// TwinCAT 3 PLC project mobject_core
// Title: mobject-core
// Company: mobject.io
// Author: mobject dev team
// ProjectVersion: 0.9.0
// ProgramVersion: 3.1.4023.0
// libraries:
//   Tc2_Standard, * (Beckhoff Automation GmbH)
//   Tc2_System, * (Beckhoff Automation GmbH)
//   Tc2_Utilities, * (Beckhoff Automation GmbH)
//   Tc3_DynamicMemory, * (Beckhoff Automation GmbH)
//   Tc3_Module, * (Beckhoff Automation GmbH)
// project tree:
//   Command/By Inheritance/ Command.TcPOU
//   Command/ I_Command.TcIO
//   / Constants.TcGVL
//   Cyclic Instance/By Composition/ AutomaticCyclicCall.TcPOU, ManualCyclicCall.TcPOU
//   Cyclic Instance/By Inheritance/ CyclicInstance.TcPOU
//   Cyclic Instance/ I_CyclicInstance.TcIO (not stored)
//   Functions/Command Feedback/ F_IsError.TcPOU, F_IsDone.TcPOU, F_IsBusy.TcPOU, F_GetErrorId.TcPOU
//   Functions/Converters/BOOL_TO_/ Convert_BOOL_TO_.TcPOU (not stored), Convert_BOOL_TO_BOOL.TcPOU (not stored), Convert_BOOL_TO_BYTE.TcPOU, Convert_BOOL_TO_DATE.TcPOU, Convert_BOOL_TO_DINT.TcPOU, Convert_BOOL_TO_DT.TcPOU (not stored), Convert_BOOL_TO_DWORD.TcPOU (not stored), Convert_BOOL_TO_INT.TcPOU (not stored), Convert_BOOL_TO_LINT.TcPOU (not stored), Convert_BOOL_TO_LREAL.TcPOU, Convert_BOOL_TO_LWORD.TcPOU, Convert_BOOL_TO_REAL.TcPOU (not stored), Convert_BOOL_TO_SINT.TcPOU, Convert_BOOL_TO_STRING.TcPOU (not stored), Convert_BOOL_TO_TIME.TcPOU, Convert_BOOL_TO_TOD.TcPOU, Convert_BOOL_TO_UDINT.TcPOU (not stored), Convert_BOOL_TO_UINT.TcPOU, Convert_BOOL_TO_ULINT.TcPOU, Convert_BOOL_TO_USINT.TcPOU (not stored), Convert_BOOL_TO_WORD.TcPOU
//   Functions/Converters/BYTE_TO_/ Convert_BYTE_TO_.TcPOU (not stored), Convert_BYTE_TO_BOOL.TcPOU (not stored), Convert_BYTE_TO_BYTE.TcPOU, Convert_BYTE_TO_DATE.TcPOU, Convert_BYTE_TO_DINT.TcPOU (not stored), Convert_BYTE_TO_DT.TcPOU, Convert_BYTE_TO_DWORD.TcPOU (not stored), Convert_BYTE_TO_INT.TcPOU (not stored), Convert_BYTE_TO_LINT.TcPOU (not stored), Convert_BYTE_TO_LREAL.TcPOU, Convert_BYTE_TO_LWORD.TcPOU (not stored), Convert_BYTE_TO_REAL.TcPOU, Convert_BYTE_TO_SINT.TcPOU (not stored), Convert_BYTE_TO_STRING.TcPOU (not stored), Convert_BYTE_TO_TIME.TcPOU, Convert_BYTE_TO_TOD.TcPOU (not stored), Convert_BYTE_TO_UDINT.TcPOU, Convert_BYTE_TO_UINT.TcPOU, Convert_BYTE_TO_ULINT.TcPOU, Convert_BYTE_TO_USINT.TcPOU (not stored), Convert_BYTE_TO_WORD.TcPOU
//   Functions/Converters/DATE_TO_/ Convert_DATE_TO_.TcPOU, Convert_DATE_TO_BOOL.TcPOU, Convert_DATE_TO_BYTE.TcPOU, Convert_DATE_TO_DATE.TcPOU, Convert_DATE_TO_DINT.TcPOU, Convert_DATE_TO_DT.TcPOU (not stored), Convert_DATE_TO_DWORD.TcPOU (not stored), Convert_DATE_TO_INT.TcPOU, Convert_DATE_TO_LINT.TcPOU (not stored), Convert_DATE_TO_LREAL.TcPOU (not stored), Convert_DATE_TO_LWORD.TcPOU (not stored), Convert_DATE_TO_REAL.TcPOU, Convert_DATE_TO_SINT.TcPOU, Convert_DATE_TO_STRING.TcPOU, Convert_DATE_TO_TIME.TcPOU, Convert_DATE_TO_TOD.TcPOU, Convert_DATE_TO_UDINT.TcPOU, Convert_DATE_TO_UINT.TcPOU (not stored), Convert_DATE_TO_ULINT.TcPOU (not stored), Convert_DATE_TO_USINT.TcPOU (not stored), Convert_DATE_TO_WORD.TcPOU
//   Functions/Converters/DINT_TO_/ Convert_DINT_TO_.TcPOU, Convert_DINT_TO_BOOL.TcPOU, Convert_DINT_TO_BYTE.TcPOU, Convert_DINT_TO_DATE.TcPOU (not stored), Convert_DINT_TO_DINT.TcPOU (not stored), Convert_DINT_TO_DT.TcPOU (not stored), Convert_DINT_TO_DWORD.TcPOU, Convert_DINT_TO_INT.TcPOU, Convert_DINT_TO_LINT.TcPOU, Convert_DINT_TO_LREAL.TcPOU (not stored), Convert_DINT_TO_LWORD.TcPOU, Convert_DINT_TO_REAL.TcPOU (not stored), Convert_DINT_TO_SINT.TcPOU, Convert_DINT_TO_STRING.TcPOU, Convert_DINT_TO_TIME.TcPOU (not stored), Convert_DINT_TO_TOD.TcPOU (not stored), Convert_DINT_TO_UDINT.TcPOU, Convert_DINT_TO_UINT.TcPOU (not stored), Convert_DINT_TO_ULINT.TcPOU (not stored), Convert_DINT_TO_USINT.TcPOU, Convert_DINT_TO_WORD.TcPOU
//   Functions/Converters/DT_TO_/ Convert_DT_TO_.TcPOU (not stored), Convert_DT_TO_BOOL.TcPOU, Convert_DT_TO_BYTE.TcPOU, Convert_DT_TO_DATE.TcPOU, Convert_DT_TO_DINT.TcPOU (not stored), Convert_DT_TO_DT.TcPOU (not stored), Convert_DT_TO_DWORD.TcPOU, Convert_DT_TO_INT.TcPOU, Convert_DT_TO_LINT.TcPOU (not stored), Convert_DT_TO_LREAL.TcPOU (not stored), Convert_DT_TO_LWORD.TcPOU, Convert_DT_TO_REAL.TcPOU, Convert_DT_TO_SINT.TcPOU, Convert_DT_TO_STRING.TcPOU, Convert_DT_TO_TIME.TcPOU (not stored), Convert_DT_TO_TOD.TcPOU (not stored), Convert_DT_TO_UDINT.TcPOU, Convert_DT_TO_UINT.TcPOU, Convert_DT_TO_ULINT.TcPOU (not stored), Convert_DT_TO_USINT.TcPOU, Convert_DT_TO_WORD.TcPOU (not stored)
//   Functions/Converters/DWORD_TO_/ Convert_DWORD_TO_.TcPOU, Convert_DWORD_TO_BOOL.TcPOU (not stored), Convert_DWORD_TO_BYTE.TcPOU, Convert_DWORD_TO_DATE.TcPOU, Convert_DWORD_TO_DINT.TcPOU (not stored), Convert_DWORD_TO_DT.TcPOU (not stored), Convert_DWORD_TO_DWORD.TcPOU, Convert_DWORD_TO_INT.TcPOU, Convert_DWORD_TO_LINT.TcPOU, Convert_DWORD_TO_LREAL.TcPOU (not stored), Convert_DWORD_TO_LWORD.TcPOU, Convert_DWORD_TO_REAL.TcPOU, Convert_DWORD_TO_SINT.TcPOU (not stored), Convert_DWORD_TO_STRING.TcPOU (not stored), Convert_DWORD_TO_TIME.TcPOU (not stored), Convert_DWORD_TO_TOD.TcPOU, Convert_DWORD_TO_UDINT.TcPOU, Convert_DWORD_TO_UINT.TcPOU, Convert_DWORD_TO_ULINT.TcPOU, Convert_DWORD_TO_USINT.TcPOU (not stored), Convert_DWORD_TO_WORD.TcPOU
//   Functions/Converters/INT_TO_/ Convert_INT_TO_.TcPOU (not stored), Convert_INT_TO_BOOL.TcPOU (not stored), Convert_INT_TO_BYTE.TcPOU, Convert_INT_TO_DATE.TcPOU (not stored), Convert_INT_TO_DINT.TcPOU (not stored), Convert_INT_TO_DT.TcPOU, Convert_INT_TO_DWORD.TcPOU (not stored), Convert_INT_TO_INT.TcPOU (not stored), Convert_INT_TO_LINT.TcPOU (not stored), Convert_INT_TO_LREAL.TcPOU, Convert_INT_TO_LWORD.TcPOU, Convert_INT_TO_REAL.TcPOU (not stored), Convert_INT_TO_SINT.TcPOU (not stored), Convert_INT_TO_STRING.TcPOU, Convert_INT_TO_TIME.TcPOU (not stored), Convert_INT_TO_TOD.TcPOU, Convert_INT_TO_UDINT.TcPOU (not stored), Convert_INT_TO_UINT.TcPOU (not stored), Convert_INT_TO_ULINT.TcPOU (not stored), Convert_INT_TO_USINT.TcPOU (not stored), Convert_INT_TO_WORD.TcPOU (not stored)
//   Functions/Converters/LINT_TO/ Convert_LINT_TO_.TcPOU (not stored), Convert_LINT_TO_BOOL.TcPOU (not stored), Convert_LINT_TO_BYTE.TcPOU (not stored), Convert_LINT_TO_DATE.TcPOU, Convert_LINT_TO_DINT.TcPOU (not stored), Convert_LINT_TO_DT.TcPOU (not stored), Convert_LINT_TO_DWORD.TcPOU, Convert_LINT_TO_INT.TcPOU (not stored), Convert_LINT_TO_LINT.TcPOU (not stored), Convert_LINT_TO_LREAL.TcPOU (not stored), Convert_LINT_TO_LWORD.TcPOU, Convert_LINT_TO_REAL.TcPOU, Convert_LINT_TO_SINT.TcPOU, Convert_LINT_TO_STRING.TcPOU (not stored), Convert_LINT_TO_TIME.TcPOU, Convert_LINT_TO_TOD.TcPOU (not stored), Convert_LINT_TO_UDINT.TcPOU, Convert_LINT_TO_UINT.TcPOU, Convert_LINT_TO_ULINT.TcPOU, Convert_LINT_TO_USINT.TcPOU (not stored), Convert_LINT_TO_WORD.TcPOU
//   Functions/Converters/LREAL_TO_/ Convert_LREAL_TO_.TcPOU, Convert_LREAL_TO_BOOL.TcPOU, Convert_LREAL_TO_BYTE.TcPOU, Convert_LREAL_TO_DATE.TcPOU, Convert_LREAL_TO_DINT.TcPOU (not stored), Convert_LREAL_TO_DT.TcPOU, Convert_LREAL_TO_DWORD.TcPOU, Convert_LREAL_TO_INT.TcPOU, Convert_LREAL_TO_LINT.TcPOU (not stored), Convert_LREAL_TO_LREAL.TcPOU (not stored), Convert_LREAL_TO_LWORD.TcPOU, Convert_LREAL_TO_REAL.TcPOU (not stored), Convert_LREAL_TO_SINT.TcPOU (not stored), Convert_LREAL_TO_STRING.TcPOU (not stored), Convert_LREAL_TO_TIME.TcPOU, Convert_LREAL_TO_TOD.TcPOU (not stored), Convert_LREAL_TO_UDINT.TcPOU (not stored), Convert_LREAL_TO_UINT.TcPOU, Convert_LREAL_TO_ULINT.TcPOU, Convert_LREAL_TO_USINT.TcPOU, Convert_LREAL_TO_WORD.TcPOU
//   Functions/Converters/LWORD_TO_/ Convert_LWORD_TO_.TcPOU (not stored), Convert_LWORD_TO_BOOL.TcPOU, Convert_LWORD_TO_BYTE.TcPOU (not stored), Convert_LWORD_TO_DATE.TcPOU (not stored), Convert_LWORD_TO_DINT.TcPOU (not stored), Convert_LWORD_TO_DT.TcPOU (not stored), Convert_LWORD_TO_DWORD.TcPOU (not stored), Convert_LWORD_TO_INT.TcPOU (not stored), Convert_LWORD_TO_LINT.TcPOU, Convert_LWORD_TO_LREAL.TcPOU (not stored), Convert_LWORD_TO_LWORD.TcPOU (not stored), Convert_LWORD_TO_REAL.TcPOU (not stored), Convert_LWORD_TO_SINT.TcPOU, Convert_LWORD_TO_STRING.TcPOU, Convert_LWORD_TO_TIME.TcPOU, Convert_LWORD_TO_TOD.TcPOU (not stored), Convert_LWORD_TO_UDINT.TcPOU, Convert_LWORD_TO_UINT.TcPOU, Convert_LWORD_TO_ULINT.TcPOU (not stored), Convert_LWORD_TO_USINT.TcPOU, Convert_LWORD_TO_WORD.TcPOU (not stored)
//   Functions/Converters/REAL_TO_/ Convert_REAL_TO_.TcPOU, Convert_REAL_TO_BOOL.TcPOU (not stored), Convert_REAL_TO_BYTE.TcPOU, Convert_REAL_TO_DATE.TcPOU, Convert_REAL_TO_DINT.TcPOU, Convert_REAL_TO_DT.TcPOU (not stored), Convert_REAL_TO_DWORD.TcPOU, Convert_REAL_TO_INT.TcPOU (not stored), Convert_REAL_TO_LINT.TcPOU, Convert_REAL_TO_LREAL.TcPOU (not stored), Convert_REAL_TO_LWORD.TcPOU, Convert_REAL_TO_REAL.TcPOU (not stored), Convert_REAL_TO_SINT.TcPOU (not stored), Convert_REAL_TO_STRING.TcPOU, Convert_REAL_TO_TIME.TcPOU (not stored), Convert_REAL_TO_TOD.TcPOU (not stored), Convert_REAL_TO_UDINT.TcPOU (not stored), Convert_REAL_TO_UINT.TcPOU (not stored), Convert_REAL_TO_ULINT.TcPOU (not stored), Convert_REAL_TO_USINT.TcPOU (not stored), Convert_REAL_TO_WORD.TcPOU (not stored)
//   Functions/Converters/SINT_TO_/ Convert_SINT_TO_.TcPOU (not stored), Convert_SINT_TO_BOOL.TcPOU (not stored), Convert_SINT_TO_BYTE.TcPOU (not stored), Convert_SINT_TO_DATE.TcPOU (not stored), Convert_SINT_TO_DINT.TcPOU (not stored), Convert_SINT_TO_DT.TcPOU (not stored), Convert_SINT_TO_DWORD.TcPOU (not stored), Convert_SINT_TO_INT.TcPOU (not stored), Convert_SINT_TO_LINT.TcPOU (not stored), Convert_SINT_TO_LREAL.TcPOU (not stored), Convert_SINT_TO_LWORD.TcPOU (not stored), Convert_SINT_TO_REAL.TcPOU (not stored), Convert_SINT_TO_SINT.TcPOU (not stored), Convert_SINT_TO_STRING.TcPOU (not stored), Convert_SINT_TO_TIME.TcPOU (not stored), Convert_SINT_TO_TOD.TcPOU (not stored), Convert_SINT_TO_UDINT.TcPOU (not stored), Convert_SINT_TO_UINT.TcPOU (not stored), Convert_SINT_TO_ULINT.TcPOU (not stored), Convert_SINT_TO_USINT.TcPOU (not stored), Convert_SINT_TO_WORD.TcPOU (not stored)
//   Functions/Converters/STRING_TO_/ Convert_STRING_TO_.TcPOU (not stored), Convert_STRING_TO_BOOL.TcPOU (not stored), Convert_STRING_TO_BYTE.TcPOU (not stored), Convert_STRING_TO_DATE.TcPOU (not stored), Convert_STRING_TO_DINT.TcPOU (not stored), Convert_STRING_TO_DT.TcPOU (not stored), Convert_STRING_TO_DWORD.TcPOU (not stored), Convert_STRING_TO_INT.TcPOU (not stored), Convert_STRING_TO_LINT.TcPOU (not stored), Convert_STRING_TO_LREAL.TcPOU (not stored), Convert_STRING_TO_LWORD.TcPOU (not stored), Convert_STRING_TO_REAL.TcPOU (not stored), Convert_STRING_TO_SINT.TcPOU (not stored), Convert_STRING_TO_STRING.TcPOU (not stored), Convert_STRING_TO_TIME.TcPOU (not stored), Convert_STRING_TO_TOD.TcPOU (not stored), Convert_STRING_TO_UDINT.TcPOU (not stored), Convert_STRING_TO_UINT.TcPOU (not stored), Convert_STRING_TO_ULINT.TcPOU (not stored), Convert_STRING_TO_USINT.TcPOU (not stored), Convert_STRING_TO_WORD.TcPOU (not stored)
//   Functions/Converters/TIME_TO_/ Convert_TIME_TO_.TcPOU (not stored), Convert_TIME_TO_BOOL.TcPOU (not stored), Convert_TIME_TO_BYTE.TcPOU (not stored), Convert_TIME_TO_DATE.TcPOU (not stored), Convert_TIME_TO_DINT.TcPOU (not stored), Convert_TIME_TO_DT.TcPOU (not stored), Convert_TIME_TO_DWORD.TcPOU (not stored), Convert_TIME_TO_INT.TcPOU (not stored), Convert_TIME_TO_LINT.TcPOU (not stored), Convert_TIME_TO_LREAL.TcPOU (not stored), Convert_TIME_TO_LWORD.TcPOU (not stored), Convert_TIME_TO_REAL.TcPOU (not stored), Convert_TIME_TO_SINT.TcPOU (not stored), Convert_TIME_TO_STRING.TcPOU (not stored), Convert_TIME_TO_TIME.TcPOU (not stored), Convert_TIME_TO_TOD.TcPOU (not stored), Convert_TIME_TO_UDINT.TcPOU (not stored), Convert_TIME_TO_UINT.TcPOU (not stored), Convert_TIME_TO_ULINT.TcPOU (not stored), Convert_TIME_TO_USINT.TcPOU (not stored), Convert_TIME_TO_WORD.TcPOU (not stored)
//   Functions/Converters/TOD_TO_/ Convert_TOD_TO_.TcPOU (not stored), Convert_TOD_TO_BOOL.TcPOU (not stored), Convert_TOD_TO_BYTE.TcPOU (not stored), Convert_TOD_TO_DATE.TcPOU (not stored), Convert_TOD_TO_DINT.TcPOU (not stored), Convert_TOD_TO_DT.TcPOU (not stored), Convert_TOD_TO_DWORD.TcPOU (not stored), Convert_TOD_TO_INT.TcPOU (not stored), Convert_TOD_TO_LINT.TcPOU (not stored), Convert_TOD_TO_LREAL.TcPOU (not stored), Convert_TOD_TO_LWORD.TcPOU (not stored), Convert_TOD_TO_REAL.TcPOU (not stored), Convert_TOD_TO_SINT.TcPOU (not stored), Convert_TOD_TO_STRING.TcPOU (not stored), Convert_TOD_TO_TIME.TcPOU (not stored), Convert_TOD_TO_TOD.TcPOU (not stored), Convert_TOD_TO_UDINT.TcPOU (not stored), Convert_TOD_TO_UINT.TcPOU (not stored), Convert_TOD_TO_ULINT.TcPOU (not stored), Convert_TOD_TO_USINT.TcPOU (not stored), Convert_TOD_TO_WORD.TcPOU (not stored)
//   Functions/Converters/UDINT_TO_/ Convert_UDINT_TO_.TcPOU (not stored), Convert_UDINT_TO_BOOL.TcPOU (not stored), Convert_UDINT_TO_BYTE.TcPOU (not stored), Convert_UDINT_TO_DATE.TcPOU (not stored), Convert_UDINT_TO_DINT.TcPOU (not stored), Convert_UDINT_TO_DT.TcPOU (not stored), Convert_UDINT_TO_DWORD.TcPOU (not stored), Convert_UDINT_TO_INT.TcPOU (not stored), Convert_UDINT_TO_LINT.TcPOU (not stored), Convert_UDINT_TO_LREAL.TcPOU (not stored), Convert_UDINT_TO_LWORD.TcPOU (not stored), Convert_UDINT_TO_REAL.TcPOU (not stored), Convert_UDINT_TO_SINT.TcPOU (not stored), Convert_UDINT_TO_STRING.TcPOU (not stored), Convert_UDINT_TO_TIME.TcPOU (not stored), Convert_UDINT_TO_TOD.TcPOU (not stored), Convert_UDINT_TO_UDINT.TcPOU (not stored), Convert_UDINT_TO_UINT.TcPOU (not stored), Convert_UDINT_TO_ULINT.TcPOU (not stored), Convert_UDINT_TO_USINT.TcPOU (not stored), Convert_UDINT_TO_WORD.TcPOU (not stored)
//   Functions/Converters/UINT_TO_/ Convert_UINT_TO_.TcPOU (not stored), Convert_UINT_TO_BOOL.TcPOU (not stored), Convert_UINT_TO_BYTE.TcPOU (not stored), Convert_UINT_TO_DATE.TcPOU (not stored), Convert_UINT_TO_DINT.TcPOU (not stored), Convert_UINT_TO_DT.TcPOU (not stored), Convert_UINT_TO_DWORD.TcPOU (not stored), Convert_UINT_TO_INT.TcPOU (not stored), Convert_UINT_TO_LINT.TcPOU (not stored), Convert_UINT_TO_LREAL.TcPOU (not stored), Convert_UINT_TO_LWORD.TcPOU (not stored), Convert_UINT_TO_REAL.TcPOU (not stored), Convert_UINT_TO_SINT.TcPOU (not stored), Convert_UINT_TO_STRING.TcPOU (not stored), Convert_UINT_TO_TIME.TcPOU (not stored), Convert_UINT_TO_TOD.TcPOU (not stored), Convert_UINT_TO_UDINT.TcPOU (not stored), Convert_UINT_TO_UINT.TcPOU (not stored), Convert_UINT_TO_ULINT.TcPOU (not stored), Convert_UINT_TO_USINT.TcPOU (not stored), Convert_UINT_TO_WORD.TcPOU (not stored)
//   Functions/Converters/ULINT_TO_/ Convert_ULINT_TO_.TcPOU (not stored), Convert_ULINT_TO_BOOL.TcPOU (not stored), Convert_ULINT_TO_BYTE.TcPOU (not stored), Convert_ULINT_TO_DATE.TcPOU (not stored), Convert_ULINT_TO_DINT.TcPOU (not stored), Convert_ULINT_TO_DT.TcPOU (not stored), Convert_ULINT_TO_DWORD.TcPOU (not stored), Convert_ULINT_TO_INT.TcPOU (not stored), Convert_ULINT_TO_LINT.TcPOU (not stored), Convert_ULINT_TO_LREAL.TcPOU (not stored), Convert_ULINT_TO_LWORD.TcPOU (not stored), Convert_ULINT_TO_REAL.TcPOU (not stored), Convert_ULINT_TO_SINT.TcPOU (not stored), Convert_ULINT_TO_STRING.TcPOU (not stored), Convert_ULINT_TO_TIME.TcPOU (not stored), Convert_ULINT_TO_TOD.TcPOU (not stored), Convert_ULINT_TO_UDINT.TcPOU (not stored), Convert_ULINT_TO_UINT.TcPOU (not stored), Convert_ULINT_TO_ULINT.TcPOU (not stored), Convert_ULINT_TO_USINT.TcPOU (not stored), Convert_ULINT_TO_WORD.TcPOU (not stored)
//   Functions/Converters/USINT_TO_/ Convert_USINT_TO_.TcPOU (not stored), Convert_USINT_TO_BOOL.TcPOU (not stored), Convert_USINT_TO_BYTE.TcPOU (not stored), Convert_USINT_TO_DATE.TcPOU (not stored), Convert_USINT_TO_DINT.TcPOU (not stored), Convert_USINT_TO_DT.TcPOU (not stored), Convert_USINT_TO_DWORD.TcPOU (not stored), Convert_USINT_TO_INT.TcPOU (not stored), Convert_USINT_TO_LINT.TcPOU (not stored), Convert_USINT_TO_LREAL.TcPOU (not stored), Convert_USINT_TO_LWORD.TcPOU (not stored), Convert_USINT_TO_REAL.TcPOU (not stored), Convert_USINT_TO_SINT.TcPOU (not stored), Convert_USINT_TO_STRING.TcPOU (not stored), Convert_USINT_TO_TIME.TcPOU (not stored), Convert_USINT_TO_TOD.TcPOU (not stored), Convert_USINT_TO_UDINT.TcPOU (not stored), Convert_USINT_TO_UINT.TcPOU (not stored), Convert_USINT_TO_ULINT.TcPOU (not stored), Convert_USINT_TO_USINT.TcPOU (not stored), Convert_USINT_TO_WORD.TcPOU (not stored)
//   Functions/Converters/WORD_TO_/ Convert_WORD_TO_.TcPOU (not stored), Convert_WORD_TO_BOOL.TcPOU (not stored), Convert_WORD_TO_BYTE.TcPOU (not stored), Convert_WORD_TO_DATE.TcPOU (not stored), Convert_WORD_TO_DINT.TcPOU (not stored), Convert_WORD_TO_DT.TcPOU (not stored), Convert_WORD_TO_DWORD.TcPOU (not stored), Convert_WORD_TO_INT.TcPOU (not stored), Convert_WORD_TO_LINT.TcPOU (not stored), Convert_WORD_TO_LREAL.TcPOU (not stored), Convert_WORD_TO_LWORD.TcPOU (not stored), Convert_WORD_TO_REAL.TcPOU (not stored), Convert_WORD_TO_SINT.TcPOU (not stored), Convert_WORD_TO_STRING.TcPOU (not stored), Convert_WORD_TO_TIME.TcPOU (not stored), Convert_WORD_TO_TOD.TcPOU (not stored), Convert_WORD_TO_UDINT.TcPOU (not stored), Convert_WORD_TO_UINT.TcPOU (not stored), Convert_WORD_TO_ULINT.TcPOU (not stored), Convert_WORD_TO_USINT.TcPOU (not stored), Convert_WORD_TO_WORD.TcPOU (not stored)
//   Functions/Disposable/ F_SafeRelease.TcPOU
//   _Internal/Collections/ Collection.TcPOU, CollectionNode.TcPOU, I_Collectable.TcIO, I_CollectionNode.TcIO
//   _Internal/CommandFeedback/ CommandFeedback.TcPOU, I_CommandAbortingState.TcIO, I_CommandBusyState.TcIO, I_CommandFeedback.TcIO, I_CommandFeedbackReadWrite.TcIO
//   _Internal/Command/ I_CanReleaseWhenDone.TcIO
//   _Internal/CyclicCallback/Base/ CyclicCallback.TcPOU (not stored)
//   _Internal/CyclicCallback/Interface/ I_CyclicCalled.TcIO (not stored)
//   _Internal/Disposable/ Disposable.TcPOU, I_Disposable.TcIO
//   _Internal/Events/Base/ Event.TcPOU (not stored), I_Event.TcIO (not stored)
//   _Internal/Events/Collections/ SubscriberCollection.TcPOU (not stored)
//   _Internal/Events/Interfaces/ I_Callback.TcIO (not stored), I_Subscriber.TcIO (not stored)
//   _Internal/Functions/Namespace/ ReturnNamespaceFromInstancePath.TcPOU (not stored), ReturnSubSectionFromInstancePath.TcPOU (not stored)
//   _Internal/GlobalInstanceMembership/ GlobalInstanceMembership.TcPOU
//   _Internal/GlobalInstancesMembers/ GlobalInstanceMembers.TcPOU
//   _Internal/GlobalNamespace/ GlobalNamespace.TcPOU
//   _Internal/Instance/Collection/ InstanceCollection.TcPOU (not stored)
//   _Internal/Instance/Events/InstanceAdded/ InstanceAddedEvent.TcPOU (not stored), I_InstanceAddedEvent.TcIO (not stored)
//   _Internal/Instance/Events/InstanceRemoved/ InstanceRemovedEvent.TcPOU (not stored), I_InstanceRemovedEvent.TcIO (not stored)
//   _Internal/Instance/ Instance.TcPOU, I_Instance.TcIO
//   _Internal/Task/Callbacks/ DeregisterInstanceFromTaskCallback.TcPOU (not stored), RegisterInstanceToTaskCallback.TcPOU (not stored)
//   _Internal/Task/Events/TaskCyclicEvent/ I_TaskCyclicEvent.TcIO (not stored), TaskCyclicEvent.TcPOU (not stored)
//   _Internal/Task/Visitors/ I_VisitIntances.TcIO (not stored), RegisterInstancesToTaskVisitor.TcPOU (not stored)
//   Task/ I_Task.TcIO, Task.TcPOU

// ---- Constants.TcGVL
VAR_GLOBAL CONSTANT
	INVALIDPARM : HRESULT := UDINT_TO_DINT(16#9811070B);
	NOT_FOUND : HRESULT := UDINT_TO_DINT(16#9811070C);
	INCOMPATIBLE : HRESULT := UDINT_TO_DINT(16#9811070E);
END_VAR

// ---- Command/I_Command.TcIO
INTERFACE I_Command EXTENDS I_Disposable

METHOD PUBLIC Abort : I_CanReleaseWhenDone
VAR_INPUT
END_VAR
END_METHOD

METHOD PUBLIC Execute : I_CanReleaseWhenDone
VAR_INPUT
	Feedback : REFERENCE TO I_CommandFeedback;
END_VAR
END_METHOD

END_INTERFACE

// ---- _Internal/Collections/I_Collectable.TcIO
INTERFACE I_Collectable EXTENDS __SYSTEM.IQueryInterface

END_INTERFACE

// ---- _Internal/Collections/I_CollectionNode.TcIO
INTERFACE I_CollectionNode

PROPERTY PUBLIC Collectable : I_Collectable
GET
END_GET
END_PROPERTY

METHOD PUBLIC Destroy
VAR_INPUT
END_VAR
END_METHOD

PROPERTY PUBLIC Next : I_CollectionNode
GET
END_GET
SET
END_SET
END_PROPERTY

END_INTERFACE

// ---- _Internal/CommandFeedback/I_CommandAbortingState.TcIO
INTERFACE I_CommandAbortingState

METHOD PUBLIC SetAborted
VAR_INPUT
END_VAR
END_METHOD

METHOD PUBLIC SetError
VAR_INPUT
	ErrorId : UDINT;
END_VAR
END_METHOD

END_INTERFACE

// ---- _Internal/CommandFeedback/I_CommandBusyState.TcIO
INTERFACE I_CommandBusyState

METHOD PUBLIC SetAborting
VAR_INPUT
END_VAR
END_METHOD

METHOD PUBLIC SetDone
VAR_INPUT
END_VAR
END_METHOD

METHOD PUBLIC SetError
VAR_INPUT
	ErrorId : UDINT;
END_VAR
END_METHOD

END_INTERFACE

// ---- _Internal/CommandFeedback/I_CommandFeedback.TcIO
INTERFACE I_CommandFeedback EXTENDS I_Disposable

PROPERTY Aborted : BOOL
GET
END_GET
END_PROPERTY

PROPERTY Aborting : BOOL
GET
END_GET
END_PROPERTY

PROPERTY Busy : BOOL
GET
END_GET
END_PROPERTY

PROPERTY Done : BOOL
GET
END_GET
END_PROPERTY

PROPERTY Error : BOOL
GET
END_GET
END_PROPERTY

PROPERTY PUBLIC ErrorId : UDINT
GET
END_GET
END_PROPERTY

END_INTERFACE

// ---- _Internal/CommandFeedback/I_CommandFeedbackReadWrite.TcIO
INTERFACE I_CommandFeedbackReadWrite EXTENDS I_CommandFeedback, I_CommandBusyState, I_CommandAbortingState

METHOD PUBLIC SetBusy
VAR_INPUT
END_VAR
END_METHOD

END_INTERFACE

// ---- _Internal/Command/I_CanReleaseWhenDone.TcIO
INTERFACE I_CanReleaseWhenDone

METHOD PUBLIC ThenRelease
VAR_INPUT
END_VAR
END_METHOD

END_INTERFACE

// ---- _Internal/Disposable/I_Disposable.TcIO
INTERFACE I_Disposable EXTENDS __SYSTEM.IQueryInterface

METHOD AddReference
VAR_INPUT
END_VAR
END_METHOD

METHOD Release
VAR_INPUT
END_VAR
END_METHOD

END_INTERFACE

// ---- _Internal/Instance/I_Instance.TcIO
INTERFACE I_Instance EXTENDS I_Collectable

PROPERTY PUBLIC NameSpace : STRING
GET
END_GET
END_PROPERTY

METHOD PUBLIC SharesNamespaceWith : BOOL
VAR_INPUT
	OtherInstance : I_Instance;
END_VAR
END_METHOD

END_INTERFACE

// ---- Task/I_Task.TcIO
INTERFACE I_Task EXTENDS I_Instance

METHOD PUBLIC CyclicCall
END_METHOD

METHOD PUBLIC DeregisterInstance
VAR_INPUT
	Instance : I_Instance;
END_VAR
END_METHOD

PROPERTY PUBLIC Index : DINT
GET
END_GET
END_PROPERTY

PROPERTY Info : reference to PlcTaskSystemInfo
GET
END_GET
END_PROPERTY

METHOD PUBLIC IsExecutingThis : BOOL
VAR_INPUT
END_VAR
END_METHOD

PROPERTY PUBLIC OnCyclicCall : I_Event
GET
END_GET
END_PROPERTY

METHOD PUBLIC RegisterInstance
VAR_INPUT
	Instance : I_Instance;
END_VAR
END_METHOD

END_INTERFACE

// ---- Command/By Inheritance/Command.TcPOU
{attribute 'linkalways'} 
{attribute 'no_explicit_call' := 'This FB is a CLASS and must be accessed using methods or properties'}
{attribute 'enable_dynamic_creation'}
FUNCTION_BLOCK ABSTRACT Command EXTENDS Disposable IMPLEMENTS I_CyclicCalled, I_Command, I_CanReleaseWhenDone
VAR
	cyclicCall : ManualCyclicCall(THIS^);
	commandFeedback : I_CommandFeedbackReadWrite;
	commandHasCompleted : BOOL;
	disposeOnceComplete : BOOL;
END_VAR

METHOD PUBLIC Abort : I_CanReleaseWhenDone
VAR_INPUT
END_VAR
Abort := THIS^;

IF IsAborting() THEN
	RETURN;
END_IF

IF HasCompleted() THEN
	RETURN;
END_IF

commandFeedback.SetAborting();

OnAbort(commandFeedback);

IF HasCompleted() THEN
	DisableCyclicCalling();
	CompleteTheCommand();
	RETURN;
END_IF
END_METHOD

METHOD PRIVATE ClearFeedback
VAR_INPUT
END_VAR
commandFeedback.Release();
commandFeedback := 0;
END_METHOD

METHOD PRIVATE CompleteTheCommand
VAR_INPUT
END_VAR
ClearFeedback();

IF disposeOnceComplete THEN
	DisposeCommand();	
END_IF

OnExecuteComplete();

commandHasCompleted := TRUE;
END_METHOD

METHOD PUBLIC CyclicCall
VAR_INPUT
END_VAR
IF IsStillBusyExecuting() THEN
	WhileBusy(commandFeedback);
END_IF

IF IsAborting() THEN
	WhileAborting(commandFeedback);
END_IF

IF NOT HasCompleted() THEN 
	RETURN;
END_IF

DisableCyclicCalling();
CompleteTheCommand();
END_METHOD

METHOD PRIVATE DisableCyclicCalling
cyclicCall.Disable();
END_METHOD

METHOD PRIVATE DisposeCommand
VAR_INPUT
END_VAR
disposeOnceComplete := FALSE;

SUPER^.OnDispose();
END_METHOD

METHOD PRIVATE EnableCyclicCalling
cyclicCall.Enable();
END_METHOD

METHOD PUBLIC Execute : I_CanReleaseWhenDone
VAR_INPUT
	Feedback : REFERENCE TO I_CommandFeedback;
END_VAR
Execute := THIS^;

IF feedback <> 0 THEN 
	feedback.Release();
END_IF

IF IsAlreadyExecuting() THEN

	IF __ISVALIDREF(feedback) THEN
		feedback := commandFeedback;
		feedback.AddReference();
	END_IF
	
	RETURN;
	
END_IF

IF commandFeedback <> 0 THEN 
	commandFeedback.Release();
END_IF

commandFeedback := GetCustomFeedback();

IF commandFeedback = 0 THEN
	commandFeedback := GetStandardFeedback();
END_IF

IF __ISVALIDREF(feedback) THEN
	feedback := commandFeedback;
	feedback.AddReference();
END_IF

commandFeedback.SetBusy();

OnExecute(commandFeedback);

IF HasCompleted() THEN
	CompleteTheCommand();
	RETURN;
END_IF

EnableCyclicCalling();
END_METHOD

METHOD PROTECTED GetCustomFeedback : I_CommandFeedbackReadWrite
VAR
END_VAR
END_METHOD

METHOD PROTECTED GetStandardFeedback : I_CommandFeedbackReadWrite
VAR
	feedback : POINTER TO CommandFeedback;
END_VAR
feedback := __NEW(CommandFeedback);
GetStandardFeedback := feedback^;
END_METHOD

METHOD PRIVATE HasCompleted : BOOL
IF commandFeedback = 0 THEN
	HasCompleted := commandHasCompleted;
	RETURN;
END_IF

HasCompleted := not commandFeedback.Busy;
END_METHOD

METHOD PRIVATE IsAborting : BOOL
IF commandFeedback = 0 THEN
	RETURN;
END_IF

IsAborting := commandFeedback.Aborting;
END_METHOD

METHOD PRIVATE IsAlreadyExecuting : BOOL
IF commandFeedback = 0 THEN
	RETURN;
END_IF

IsAlreadyExecuting := commandFeedback.Busy;
END_METHOD

METHOD PRIVATE IsStillBusyExecuting : BOOL
IF commandFeedback = 0 THEN
	RETURN;
END_IF

IsStillBusyExecuting := commandFeedback.Busy and not commandFeedback.Aborting;
END_METHOD

METHOD PROTECTED OnAbort
VAR_INPUT
	CommandState : I_CommandAbortingState;
END_VAR
// override this method when a command needs time to "abort".
// if your aborting code take more than one cycle to completed then do not SetAborted() here, rather use SetAborted inside WhileAborting.
CommandState.SetAborted();
END_METHOD

METHOD PROTECTED OnDispose
VAR_INPUT
END_VAR
IF IsAlreadyExecuting() THEN 
	disposeOnceComplete := TRUE;
	Abort();
	RETURN;	
END_IF

DisposeCommand();
END_METHOD

METHOD PROTECTED OnExecute
VAR_INPUT
	CommandState : I_CommandBusyState;
END_VAR
END_METHOD

METHOD PROTECTED OnExecuteComplete
VAR_INPUT
END_VAR
END_METHOD

METHOD PUBLIC ThenRelease
VAR_INPUT
END_VAR
IF HasCompleted() THEN
	DisposeCommand();
	RETURN;
END_IF

disposeOnceComplete := true;
END_METHOD

METHOD PROTECTED WhileAborting
VAR_INPUT
	CommandState : I_CommandAbortingState;
END_VAR
// you must override both OnAbort and WhileAborting to use this method.
// if SetAborted has not been called during OnAbort then this method will be cyclically called until you do;
CommandState.SetAborted();
END_METHOD

METHOD PROTECTED ABSTRACT WhileBusy
VAR_INPUT
	CommandState : I_CommandBusyState;
END_VAR
// This will be called cyclically until the command has finished executing.  
// once done use the command below to complete the execute state.
//commandState.SetDone();

// use SetError to cancel the command.
//CommandState.SetError(ErrorID:=0);
END_METHOD

END_FUNCTION_BLOCK

// ---- _Internal/Disposable/Disposable.TcPOU
{attribute 'linkalways'} 
{attribute 'no_explicit_call' := 'This FB is a CLASS and must be accessed using methods or properties'}
{attribute 'enable_dynamic_creation'}
{attribute 'reflection'}
FUNCTION_BLOCK Disposable IMPLEMENTS I_Disposable
VAR
	{attribute 'instance-path'} 
    {attribute 'noinit'} 
	instancePathUsedToCheckIfDynamic : T_MAXSTRING;
	referenceCount : UDINT := 1;
END_VAR

METHOD AddReference
VAR_INPUT
END_VAR
VAR
	debug : UDINT;
END_VAR
referenceCount := referenceCount + 1;

debug := referenceCount;
END_METHOD

METHOD PROTECTED OnDispose
VAR_INPUT
END_VAR
__DELETE(THIS);
END_METHOD

METHOD Release
VAR_INPUT
END_VAR
VAR
	debug : UDINT;
END_VAR
referenceCount := referenceCount - 1;

debug := referenceCount;

IF referenceCount > 0 THEN
	RETURN;
END_IF

OnDispose();
END_METHOD

END_FUNCTION_BLOCK

// ---- _Internal/Instance/Instance.TcPOU
{attribute 'linkalways'} 
{attribute 'no_explicit_call' := 'This FB is a CLASS and must be accessed using methods or properties'}
{attribute 'enable_dynamic_creation'}
{attribute 'reflection'}
FUNCTION_BLOCK Instance IMPLEMENTS I_Instance, I_Collectable
{attribute 'hide_all_locals'}
VAR
	{attribute 'instance-path'} 
    {attribute 'noinit'} 
	instancePath : T_MAXSTRING;
	instanceNamespace : STRING := GetNamespace();
	globalNamespace : GlobalNamespace(THIS^);
END_VAR

METHOD PRIVATE GetNamespace : STRING
IF InstancePathIsFilled() THEN
	GetNamespace := ReturnNamespaceFromInstancePath(instancePath);
	RETURN;
END_IF

IF IsNewObjectDuringInitialization() THEN
	GetNamespace := globalNamespace.GetLastInstanceNamespace();
END_IF
END_METHOD

METHOD PRIVATE InstancePathIsFilled : BOOL
InstancePathIsFilled := instancePath <> '';
END_METHOD

METHOD PRIVATE IsNewObjectDuringInitialization : BOOL
VAR CONSTANT 
	PLC_INIT_PHASE : INT := 0;
END_VAR
IsNewObjectDuringInitialization := GETCURTASKINDEXEX() = PLC_INIT_PHASE;
END_METHOD

PROPERTY PUBLIC NameSpace : STRING
GET
Namespace := instanceNamespace;
END_GET
END_PROPERTY

METHOD PUBLIC SharesNamespaceWith : BOOL
VAR_INPUT
	OtherInstance : I_Instance;
END_VAR
SharesNamespaceWith := (Namespace = OtherInstance.NameSpace);
END_METHOD

END_FUNCTION_BLOCK

// ---- _Internal/GlobalNamespace/GlobalNamespace.TcPOU
{attribute 'linkalways'} 
{attribute 'no_explicit_call' := 'This FB is a CLASS and must be accessed using methods or properties'}
{attribute 'enable_dynamic_creation'}
FUNCTION_BLOCK GlobalNamespace
VAR_STAT // singleton
	lastInstanceNamespace : STRING;
END_VAR

METHOD FB_init : BOOL
VAR_INPUT
	bInitRetains : BOOL; // if TRUE, the retain variables are initialized (warm start / cold start)
	bInCopyCode : BOOL;  // if TRUE, the instance afterwards gets moved into the copy code (online change)
	Instance : I_Instance;
END_VAR
IF Instance.NameSpace = '' THEN
	RETURN;
END_IF

lastInstanceNamespace := Instance.NameSpace;
END_METHOD

METHOD PUBLIC GetLastInstanceNamespace : String
VAR_INPUT
END_VAR
GetLastInstanceNamespace := lastInstanceNamespace;
END_METHOD

END_FUNCTION_BLOCK

// ---- Cyclic Instance/By Composition/ManualCyclicCall.TcPOU
{attribute 'linkalways'} 
{attribute 'no_explicit_call' := 'This FB is a CLASS and must be accessed using methods or properties'}
{attribute 'enable_dynamic_creation'}
FUNCTION_BLOCK ManualCyclicCall EXTENDS Instance IMPLEMENTS I_CyclicInstance
VAR
	membership : GlobalInstanceMembership(THIS^);
	_cyclicInstanceCallback : CyclicCallback(0);
END_VAR

PROPERTY PUBLIC CyclicInstanceCallback : I_Callback
GET
CyclicInstanceCallback := _cyclicInstanceCallback;
END_GET
END_PROPERTY

METHOD PUBLIC Disable
VAR_INPUT
END_VAR
membership.Leave();
END_METHOD

METHOD PUBLIC Enable
VAR_INPUT
END_VAR
membership.Join();
END_METHOD

METHOD FB_init : BOOL
VAR_INPUT
	bInitRetains : BOOL; // if TRUE, the retain variables are initialized (warm start / cold start)
	bInCopyCode : BOOL;  // if TRUE, the instance afterwards gets moved into the copy code (online change)
	Target : I_CyclicCalled;
END_VAR
_cyclicInstanceCallback.Target := Target;
END_METHOD

END_FUNCTION_BLOCK

// ---- _Internal/GlobalInstanceMembership/GlobalInstanceMembership.TcPOU
{attribute 'linkalways'} 
{attribute 'no_explicit_call' := 'This FB is a CLASS and must be accessed using methods or properties'}
{attribute 'enable_dynamic_creation'}
FUNCTION_BLOCK GlobalInstanceMembership
VAR
	self : I_Instance;
	globalInstanceMembers : GlobalInstanceMembers;
END_VAR

METHOD FB_exit : BOOL
VAR_INPUT
	bInCopyCode : BOOL; // if TRUE, the exit method is called for exiting an instance that is copied afterwards (online change).
END_VAR
Leave();
END_METHOD

METHOD FB_init : BOOL
VAR_INPUT
	bInitRetains : BOOL; // if TRUE, the retain variables are initialized (warm start / cold start)
	bInCopyCode : BOOL;  // if TRUE, the instance afterwards gets moved into the copy code (online change)
	Self : I_Instance;
END_VAR
THIS^.self := Self;
END_METHOD

METHOD PUBLIC Join
VAR_INPUT
END_VAR
globalInstanceMembers.AddInstance(Self);
END_METHOD

METHOD PUBLIC Leave
VAR_INPUT
END_VAR
globalInstanceMembers.RemoveInstance(THIS^.self);
END_METHOD

END_FUNCTION_BLOCK

// ---- _Internal/GlobalInstancesMembers/GlobalInstanceMembers.TcPOU
{attribute 'linkalways'} 
{attribute 'no_explicit_call' := 'This FB is a CLASS and must be accessed using methods or properties'}
{attribute 'enable_dynamic_creation'}
FUNCTION_BLOCK GlobalInstanceMembers
VAR_STAT // singleton
	instances : InstanceCollection;
	instanceAddedEvent : InstanceAddedEvent;
	instanceRemovedEvent : InstanceRemovedEvent;
END_VAR

METHOD PUBLIC AddInstance
VAR_INPUT
	Instance : I_Instance;
END_VAR
IF Instance = 0 THEN
	RETURN;
END_IF

instances.Insert(Instance);
instanceAddedEvent.Notify(Instance);
END_METHOD

METHOD PUBLIC ForEachInstance
VAR_INPUT
	Visitor : I_VisitIntances;
END_VAR
VAR
	last : DINT;
	i : DINT;
END_VAR
last := instances.Count - 1;

FOR i := 0 TO last DO
	Visitor.Visit(instances.GetByIndex(i));
END_FOR
END_METHOD

PROPERTY PUBLIC OnInstanceAdded : I_Event
GET
OnInstanceAdded := instanceAddedEvent;
END_GET
END_PROPERTY

PROPERTY PUBLIC OnInstanceRemoved : I_Event
GET
OnInstanceRemoved := InstanceRemovedEvent;
END_GET
END_PROPERTY

METHOD PUBLIC RemoveInstance
VAR_INPUT
	Instance : I_Instance;
END_VAR
IF Instance = 0 THEN
	RETURN;
END_IF

instances.Remove(Instance);
InstanceRemovedEvent.Notify(Instance);
END_METHOD

END_FUNCTION_BLOCK

// ---- _Internal/CommandFeedback/CommandFeedback.TcPOU
{attribute 'linkalways'} 
{attribute 'no_explicit_call' := 'This FB is a CLASS and must be accessed using methods or properties'}
{attribute 'enable_dynamic_creation'}
FUNCTION_BLOCK CommandFeedback EXTENDS Disposable IMPLEMENTS I_CommandFeedbackReadWrite, I_CommandFeedback, I_CommandBusyState, I_CommandAbortingState
VAR
	_busy : BOOL;
	_done : BOOL;
	_aborted : BOOL;
	_aborting : BOOL;
	_error : BOOL;
	_errorId : UDINT;
END_VAR

PROPERTY Aborted : BOOL
GET
Aborted := _aborted;
END_GET
END_PROPERTY

PROPERTY Aborting : BOOL
GET
Aborting := _aborting;
END_GET
END_PROPERTY

PROPERTY Busy : BOOL
GET
Busy := _busy;
END_GET
END_PROPERTY

PROPERTY Done : BOOL
GET
Done := _done;
END_GET
END_PROPERTY

PROPERTY Error : BOOL
GET
Error := _error;
END_GET
END_PROPERTY

PROPERTY PUBLIC ErrorId : UDINT
GET
END_GET
END_PROPERTY

METHOD PUBLIC SetAborted
VAR_INPUT
END_VAR
_busy := FALSE;
_done := FALSE;
_aborted := TRUE;
_aborting := FALSE;
_error := FALSE;
_errorId := 0;
END_METHOD

METHOD PUBLIC SetAborting
VAR_INPUT
END_VAR
IF NOT Busy THEN
	SetAborted();
	RETURN;
END_IF

_busy := TRUE;
_done := FALSE;
_aborted := FALSE;
_aborting := TRUE;
_error := FALSE;
_errorId := 0;
END_METHOD

METHOD PUBLIC SetBusy
VAR_INPUT
END_VAR
_busy := TRUE;
_done := FALSE;
_aborted := FALSE;
_aborting := FALSE;
_error := FALSE;
_errorId := 0;
END_METHOD

METHOD PUBLIC SetDone
VAR_INPUT
END_VAR
_busy := FALSE;
_done := TRUE;
_aborted := FALSE;
_aborting := FALSE;
_error := FALSE;
_errorId := 0;
END_METHOD

METHOD PUBLIC SetError
VAR_INPUT
	ErrorId : UDINT;
END_VAR
_busy := FALSE;
_done := FALSE;
_aborted := FALSE;
_aborting := FALSE;
_error := TRUE;
_errorId := ErrorId;
END_METHOD

END_FUNCTION_BLOCK

// ---- Cyclic Instance/By Composition/AutomaticCyclicCall.TcPOU
{attribute 'linkalways'} 
{attribute 'no_explicit_call' := 'This FB is a CLASS and must be accessed using methods or properties'}
{attribute 'enable_dynamic_creation'}
FUNCTION_BLOCK AutomaticCyclicCall EXTENDS Instance IMPLEMENTS I_CyclicInstance
VAR
	membership : GlobalInstanceMembership(THIS^);
	_cyclicInstanceCallback : CyclicCallback(0);
END_VAR

PROPERTY PUBLIC CyclicInstanceCallback : I_Callback
GET
CyclicInstanceCallback := _cyclicInstanceCallback;
END_GET
END_PROPERTY

METHOD FB_init : BOOL
VAR_INPUT
	bInitRetains : BOOL; // if TRUE, the retain variables are initialized (warm start / cold start)
	bInCopyCode : BOOL;  // if TRUE, the instance afterwards gets moved into the copy code (online change)
	Target : I_CyclicCalled;
END_VAR
_cyclicInstanceCallback.Target := Target;
membership.Join();
END_METHOD

END_FUNCTION_BLOCK

// ---- Cyclic Instance/By Inheritance/CyclicInstance.TcPOU
{attribute 'linkalways'} 
{attribute 'no_explicit_call' := 'This FB is a CLASS and must be accessed using methods or properties'}
{attribute 'enable_dynamic_creation'}
FUNCTION_BLOCK ABSTRACT CyclicInstance EXTENDS Instance IMPLEMENTS I_CyclicCalled
VAR
	cyclicCall : AutomaticCyclicCall(THIS^);
END_VAR

METHOD ABSTRACT CyclicCall
VAR_INPUT
END_VAR
END_METHOD

END_FUNCTION_BLOCK

// ---- Functions/Command Feedback/F_IsError.TcPOU
FUNCTION F_IsError : BOOL;
VAR_INPUT
	Feedback : I_CommandFeedback;
END_VAR

IF Feedback <> 0 AND_THEN Feedback.Error THEN
	F_IsError := TRUE;
END_IF

END_FUNCTION

// ---- Functions/Command Feedback/F_IsDone.TcPOU
FUNCTION F_IsDone : BOOL;
VAR_INPUT
	Feedback : I_CommandFeedback;
END_VAR

IF Feedback <> 0 AND_THEN Feedback.Done THEN
	F_IsDone := TRUE;
END_IF

END_FUNCTION

// ---- Functions/Command Feedback/F_IsBusy.TcPOU
FUNCTION F_IsBusy : BOOL;
VAR_INPUT
	Feedback : I_CommandFeedback;
END_VAR

IF Feedback <> 0 AND_THEN Feedback.Busy THEN
	F_IsBusy := TRUE;
END_IF

END_FUNCTION

// ---- Functions/Command Feedback/F_GetErrorId.TcPOU
FUNCTION F_GetErrorId : UDINT;
VAR_INPUT
	Feedback : I_CommandFeedback;
END_VAR

IF Feedback <> 0 THEN
	F_GetErrorId := Feedback.ErrorId;
END_IF

END_FUNCTION

// ---- Functions/Converters/BOOL_TO_/Convert_BOOL_TO_BYTE.TcPOU
FUNCTION Convert_BOOL_TO_BYTE : Hresult
VAR_INPUT
	in : BOOL;
	out : REFERENCE TO BYTE;
END_VAR
VAR
	converted : BYTE;
END_VAR

converted := BOOL_TO_BYTE(in);

IF (BYTE_TO_BOOL(converted) <> in) THEN
	Convert_BOOL_TO_BYTE := INCOMPATIBLE;
	RETURN;
END_IF

out := converted;

END_FUNCTION

// ---- Functions/Converters/BOOL_TO_/Convert_BOOL_TO_DATE.TcPOU
FUNCTION Convert_BOOL_TO_DATE : Hresult
VAR_INPUT
	in : BOOL;
	out : REFERENCE TO DATE;
END_VAR
VAR
	converted : DATE;
END_VAR

converted := BOOL_TO_DATE(in);

IF (DATE_TO_BOOL(converted) <> in) THEN
	Convert_BOOL_TO_DATE := INCOMPATIBLE;
	RETURN;
END_IF

out := converted;

END_FUNCTION

// ---- Functions/Converters/BOOL_TO_/Convert_BOOL_TO_DINT.TcPOU
FUNCTION Convert_BOOL_TO_DINT : Hresult
VAR_INPUT
	in : BOOL;
	out : REFERENCE TO DINT;
END_VAR
VAR
	converted : DINT;
END_VAR

converted := BOOL_TO_DINT(in);

IF (DINT_TO_BOOL(converted) <> in) THEN
	Convert_BOOL_TO_DINT := INCOMPATIBLE;
	RETURN;
END_IF

out := converted;

END_FUNCTION

// ---- Functions/Converters/BOOL_TO_/Convert_BOOL_TO_LREAL.TcPOU
FUNCTION Convert_BOOL_TO_LREAL : Hresult
VAR_INPUT
	in : BOOL;
	out : REFERENCE TO LREAL;
END_VAR
VAR
	converted : LREAL;
END_VAR

converted := BOOL_TO_LREAL(in);

IF (LREAL_TO_BOOL(converted) <> in) THEN
	Convert_BOOL_TO_LREAL := INCOMPATIBLE;
	RETURN;
END_IF

out := converted;

END_FUNCTION

// ---- Functions/Converters/BOOL_TO_/Convert_BOOL_TO_LWORD.TcPOU
FUNCTION Convert_BOOL_TO_LWORD : Hresult
VAR_INPUT
	in : BOOL;
	out : REFERENCE TO LWORD;
END_VAR
VAR
	converted : LWORD;
END_VAR

converted := BOOL_TO_LWORD(in);

IF (LWORD_TO_BOOL(converted) <> in) THEN
	Convert_BOOL_TO_LWORD := INCOMPATIBLE;
	RETURN;
END_IF

out := converted;

END_FUNCTION

// ---- Functions/Converters/BOOL_TO_/Convert_BOOL_TO_SINT.TcPOU
FUNCTION Convert_BOOL_TO_SINT : Hresult
VAR_INPUT
	in : BOOL;
	out : REFERENCE TO SINT;
END_VAR
VAR
	converted : SINT;
END_VAR

converted := BOOL_TO_SINT(in);

IF (SINT_TO_BOOL(converted) <> in) THEN
	Convert_BOOL_TO_SINT := INCOMPATIBLE;
	RETURN;
END_IF

out := converted;

END_FUNCTION

// ---- Functions/Converters/BOOL_TO_/Convert_BOOL_TO_TIME.TcPOU
FUNCTION Convert_BOOL_TO_TIME : Hresult
VAR_INPUT
	in : BOOL;
	out : REFERENCE TO TIME;
END_VAR
VAR
	converted : TIME;
END_VAR

converted := BOOL_TO_TIME(in);

IF (TIME_TO_BOOL(converted) <> in) THEN
	Convert_BOOL_TO_TIME := INCOMPATIBLE;
	RETURN;
END_IF

out := converted;

END_FUNCTION

// ---- Functions/Converters/BOOL_TO_/Convert_BOOL_TO_TOD.TcPOU
FUNCTION Convert_BOOL_TO_TOD : Hresult
VAR_INPUT
	in : BOOL;
	out : REFERENCE TO TOD;
END_VAR
VAR
	converted : TOD;
END_VAR

converted := BOOL_TO_TOD(in);

IF (TOD_TO_BOOL(converted) <> in) THEN
	Convert_BOOL_TO_TOD := INCOMPATIBLE;
	RETURN;
END_IF

out := converted;

END_FUNCTION

// ---- Functions/Converters/BOOL_TO_/Convert_BOOL_TO_UINT.TcPOU
FUNCTION Convert_BOOL_TO_UINT : Hresult
VAR_INPUT
	in : BOOL;
	out : REFERENCE TO UINT;
END_VAR
VAR
	converted : UINT;
END_VAR

converted := BOOL_TO_UINT(in);

IF (UINT_TO_BOOL(converted) <> in) THEN
	Convert_BOOL_TO_UINT := INCOMPATIBLE;
	RETURN;
END_IF

out := converted;

END_FUNCTION

// ---- Functions/Converters/BOOL_TO_/Convert_BOOL_TO_ULINT.TcPOU
FUNCTION Convert_BOOL_TO_ULINT : Hresult
VAR_INPUT
	in : BOOL;
	out : REFERENCE TO ULINT;
END_VAR
VAR
	converted : ULINT;
END_VAR

converted := BOOL_TO_ULINT(in);

IF (ULINT_TO_BOOL(converted) <> in) THEN
	Convert_BOOL_TO_ULINT := INCOMPATIBLE;
	RETURN;
END_IF

out := converted;

END_FUNCTION

// ---- Functions/Converters/BOOL_TO_/Convert_BOOL_TO_WORD.TcPOU
FUNCTION Convert_BOOL_TO_WORD : Hresult
VAR_INPUT
	in : BOOL;
	out : REFERENCE TO WORD;
END_VAR
VAR
	converted : WORD;
END_VAR

converted := BOOL_TO_WORD(in);

IF (WORD_TO_BOOL(converted) <> in) THEN
	Convert_BOOL_TO_WORD := INCOMPATIBLE;
	RETURN;
END_IF

out := converted;

END_FUNCTION

// ---- Functions/Converters/BYTE_TO_/Convert_BYTE_TO_BYTE.TcPOU
FUNCTION Convert_BYTE_TO_BYTE : Hresult
VAR_INPUT
	in : BYTE;
	out : REFERENCE TO BYTE;
END_VAR

out := in;

END_FUNCTION

// ---- Functions/Converters/BYTE_TO_/Convert_BYTE_TO_DATE.TcPOU
FUNCTION Convert_BYTE_TO_DATE : Hresult
VAR_INPUT
	in : BYTE;
	out : REFERENCE TO DATE;
END_VAR
VAR
	converted : DATE;
END_VAR

converted := BYTE_TO_DATE(in);

IF (DATE_TO_BYTE(converted) <> in) THEN
	Convert_BYTE_TO_DATE := INCOMPATIBLE;
	RETURN;
END_IF

out := converted;

END_FUNCTION

// ---- Functions/Converters/BYTE_TO_/Convert_BYTE_TO_DT.TcPOU
FUNCTION Convert_BYTE_TO_DT : Hresult
VAR_INPUT
	in : BYTE;
	out : REFERENCE TO DT;
END_VAR
VAR
	converted : DT;
END_VAR

converted := BYTE_TO_DT(in);

IF (DT_TO_BYTE(converted) <> in) THEN
	Convert_BYTE_TO_DT := INCOMPATIBLE;
	RETURN;
END_IF

out := converted;

END_FUNCTION

// ---- Functions/Converters/BYTE_TO_/Convert_BYTE_TO_LREAL.TcPOU
FUNCTION Convert_BYTE_TO_LREAL : Hresult
VAR_INPUT
	in : BYTE;
	out : REFERENCE TO LREAL;
END_VAR
VAR
	converted : LREAL;
END_VAR

converted := BYTE_TO_LREAL(in);

IF (LREAL_TO_BYTE(converted) <> in) THEN
	Convert_BYTE_TO_LREAL := INCOMPATIBLE;
	RETURN;
END_IF

out := converted;

END_FUNCTION

// ---- Functions/Converters/BYTE_TO_/Convert_BYTE_TO_REAL.TcPOU
FUNCTION Convert_BYTE_TO_REAL : Hresult
VAR_INPUT
	in : BYTE;
	out : REFERENCE TO REAL;
END_VAR
VAR
	converted : REAL;
END_VAR

converted := BYTE_TO_REAL(in);

IF (REAL_TO_BYTE(converted) <> in) THEN
	Convert_BYTE_TO_REAL := INCOMPATIBLE;
	RETURN;
END_IF

out := converted;

END_FUNCTION

// ---- Functions/Converters/BYTE_TO_/Convert_BYTE_TO_TIME.TcPOU
FUNCTION Convert_BYTE_TO_TIME : Hresult
VAR_INPUT
	in : BYTE;
	out : REFERENCE TO TIME;
END_VAR
VAR
	converted : TIME;
END_VAR

converted := BYTE_TO_TIME(in);

IF (TIME_TO_BYTE(converted) <> in) THEN
	Convert_BYTE_TO_TIME := INCOMPATIBLE;
	RETURN;
END_IF

out := converted;

END_FUNCTION

// ---- Functions/Converters/BYTE_TO_/Convert_BYTE_TO_UDINT.TcPOU
FUNCTION Convert_BYTE_TO_UDINT : Hresult
VAR_INPUT
	in : BYTE;
	out : REFERENCE TO UDINT;
END_VAR
VAR
	converted : UDINT;
END_VAR

converted := BYTE_TO_UDINT(in);

IF (UDINT_TO_BYTE(converted) <> in) THEN
	Convert_BYTE_TO_UDINT := INCOMPATIBLE;
	RETURN;
END_IF

out := converted;

END_FUNCTION

// ---- Functions/Converters/BYTE_TO_/Convert_BYTE_TO_UINT.TcPOU
FUNCTION Convert_BYTE_TO_UINT : Hresult
VAR_INPUT
	in : BYTE;
	out : REFERENCE TO UINT;
END_VAR
VAR
	converted : UINT;
END_VAR

converted := BYTE_TO_UINT(in);

IF (UINT_TO_BYTE(converted) <> in) THEN
	Convert_BYTE_TO_UINT := INCOMPATIBLE;
	RETURN;
END_IF

out := converted;

END_FUNCTION

// ---- Functions/Converters/BYTE_TO_/Convert_BYTE_TO_ULINT.TcPOU
FUNCTION Convert_BYTE_TO_ULINT : Hresult
VAR_INPUT
	in : BYTE;
	out : REFERENCE TO ULINT;
END_VAR
VAR
	converted : ULINT;
END_VAR

converted := BYTE_TO_ULINT(in);

IF (ULINT_TO_BYTE(converted) <> in) THEN
	Convert_BYTE_TO_ULINT := INCOMPATIBLE;
	RETURN;
END_IF

out := converted;

END_FUNCTION

// ---- Functions/Converters/BYTE_TO_/Convert_BYTE_TO_WORD.TcPOU
FUNCTION Convert_BYTE_TO_WORD : Hresult
VAR_INPUT
	in : BYTE;
	out : REFERENCE TO WORD;
END_VAR
VAR
	converted : WORD;
END_VAR

converted := BYTE_TO_WORD(in);

IF (WORD_TO_BYTE(converted) <> in) THEN
	Convert_BYTE_TO_WORD := INCOMPATIBLE;
	RETURN;
END_IF

out := converted;

END_FUNCTION

// ---- Functions/Converters/DATE_TO_/Convert_DATE_TO_.TcPOU
FUNCTION Convert_DATE_TO_ : Hresult
VAR_INPUT
	in : DATE;
	out : ANY;
END_VAR
VAR
	convertResult : HRESULT := INCOMPATIBLE;
	convertAddress : PVOID;
	_BOOL : BOOL;
	_BYTE : BYTE;
	_DATE : DATE;
	_DINT : DINT;
	_DT : DT;
	_DWORD : DWORD;
	_INT : INT;
	_LINT : LINT;
	_LREAL : LREAL;
	_LWORD : LWORD;
	_REAL : REAL;
	_SINT : SINT;
	_STRING : STRING;
	_TIME : TIME;
	_TOD : TOD;
	_UDINT : UDINT;
	_UINT : UINT;
	_ULINT : ULINT;
	_USINT : USINT;
	_WORD : WORD;
END_VAR

CASE out.TypeClass OF
	
	__SYSTEM.TYPE_CLASS.TYPE_BOOL:
	
		convertResult := Convert_DATE_TO_BOOL(in, _BOOL);
		IF SUCCEEDED(convertResult) THEN
			convertAddress := ADR(_BOOL);
		END_IF

	__SYSTEM.TYPE_CLASS.TYPE_BYTE:
	
		convertResult := Convert_DATE_TO_BYTE(in, _BYTE);
		IF SUCCEEDED(convertResult) THEN
			convertAddress := ADR(_BYTE);
		END_IF

	__SYSTEM.TYPE_CLASS.TYPE_DATE:
	
		convertResult := Convert_DATE_TO_DATE(in, _DATE);
		IF SUCCEEDED(convertResult) THEN
			convertAddress := ADR(_DATE);
		END_IF

	__SYSTEM.TYPE_CLASS.TYPE_DINT:
	
		convertResult := Convert_DATE_TO_DINT(in, _DINT);
		IF SUCCEEDED(convertResult) THEN
			convertAddress := ADR(_DINT);
		END_IF

	__SYSTEM.TYPE_CLASS.TYPE_DATEANDTIME:
	
		convertResult := Convert_DATE_TO_DT(in, _DT);
		IF SUCCEEDED(convertResult) THEN
			convertAddress := ADR(_DT);
		END_IF

	__SYSTEM.TYPE_CLASS.TYPE_DWORD:
	
		convertResult := Convert_DATE_TO_DWORD(in, _DWORD);
		IF SUCCEEDED(convertResult) THEN
			convertAddress := ADR(_DWORD);
		END_IF

	__SYSTEM.TYPE_CLASS.TYPE_INT:
	
		convertResult := Convert_DATE_TO_INT(in, _INT);
		IF SUCCEEDED(convertResult) THEN
			convertAddress := ADR(_INT);
		END_IF

	__SYSTEM.TYPE_CLASS.TYPE_LINT:
	
		convertResult := Convert_DATE_TO_LINT(in, _LINT);
		IF SUCCEEDED(convertResult) THEN
			convertAddress := ADR(_LINT);
		END_IF

	__SYSTEM.TYPE_CLASS.TYPE_LREAL:
	
		convertResult := Convert_DATE_TO_LREAL(in, _LREAL);
		IF SUCCEEDED(convertResult) THEN
			convertAddress := ADR(_LREAL);
		END_IF

	__SYSTEM.TYPE_CLASS.TYPE_LWORD:
	
		convertResult := Convert_DATE_TO_LWORD(in, _LWORD);
		IF SUCCEEDED(convertResult) THEN
			convertAddress := ADR(_LWORD);
		END_IF

	__SYSTEM.TYPE_CLASS.TYPE_REAL:
	
		convertResult := Convert_DATE_TO_REAL(in, _REAL);
		IF SUCCEEDED(convertResult) THEN
			convertAddress := ADR(_REAL);
		END_IF

	__SYSTEM.TYPE_CLASS.TYPE_SINT:
	
		convertResult := Convert_DATE_TO_SINT(in, _SINT);
		IF SUCCEEDED(convertResult) THEN
			convertAddress := ADR(_SINT);
		END_IF

	__SYSTEM.TYPE_CLASS.TYPE_STRING:
	
		convertResult := Convert_DATE_TO_STRING(in, _STRING);
		IF SUCCEEDED(convertResult) THEN
			convertAddress := ADR(_STRING);
		END_IF

	__SYSTEM.TYPE_CLASS.TYPE_TIME:
	
		convertResult := Convert_DATE_TO_TIME(in, _TIME);
		IF SUCCEEDED(convertResult) THEN
			convertAddress := ADR(_TIME);
		END_IF

	__SYSTEM.TYPE_CLASS.TYPE_TIMEOFDAY:
	
		convertResult := Convert_DATE_TO_TOD(in, _TOD);
		IF SUCCEEDED(convertResult) THEN
			convertAddress := ADR(_TOD);
		END_IF

	__SYSTEM.TYPE_CLASS.TYPE_UDINT:
	
		convertResult := Convert_DATE_TO_UDINT(in, _UDINT);
		IF SUCCEEDED(convertResult) THEN
			convertAddress := ADR(_UDINT);
		END_IF

	__SYSTEM.TYPE_CLASS.TYPE_UINT:
	
		convertResult := Convert_DATE_TO_UINT(in, _UINT);
		IF SUCCEEDED(convertResult) THEN
			convertAddress := ADR(_UINT);
		END_IF

	__SYSTEM.TYPE_CLASS.TYPE_ULINT:
	
		convertResult := Convert_DATE_TO_ULINT(in, _ULINT);
		IF SUCCEEDED(convertResult) THEN
			convertAddress := ADR(_ULINT);
		END_IF

	__SYSTEM.TYPE_CLASS.TYPE_USINT:
	
		convertResult := Convert_DATE_TO_USINT(in, _USINT);
		IF SUCCEEDED(convertResult) THEN
			convertAddress := ADR(_USINT);
		END_IF

	__SYSTEM.TYPE_CLASS.TYPE_WORD:
	
		convertResult := Convert_DATE_TO_WORD(in, _WORD);
		IF SUCCEEDED(convertResult) THEN
			convertAddress := ADR(_WORD);
		END_IF

END_CASE

IF SUCCEEDED(convertResult) THEN
	memcpy(out.pValue,convertAddress,DINT_TO_UDINT(out.diSize));
END_IF

Convert_DATE_TO_ := convertResult;

END_FUNCTION

// ---- Functions/Converters/DATE_TO_/Convert_DATE_TO_BOOL.TcPOU
FUNCTION Convert_DATE_TO_BOOL : Hresult
VAR_INPUT
	in : DATE;
	out : REFERENCE TO BOOL;
END_VAR
VAR
	converted : BOOL;
END_VAR

converted := DATE_TO_BOOL(in);

IF (BOOL_TO_DATE(converted) <> in) THEN
	Convert_DATE_TO_BOOL := INCOMPATIBLE;
	RETURN;
END_IF

out := converted;

END_FUNCTION

// ---- Functions/Converters/DATE_TO_/Convert_DATE_TO_BYTE.TcPOU
FUNCTION Convert_DATE_TO_BYTE : Hresult
VAR_INPUT
	in : DATE;
	out : REFERENCE TO BYTE;
END_VAR
VAR
	converted : BYTE;
END_VAR

converted := DATE_TO_BYTE(in);

IF (BYTE_TO_DATE(converted) <> in) THEN
	Convert_DATE_TO_BYTE := INCOMPATIBLE;
	RETURN;
END_IF

out := converted;

END_FUNCTION

// ---- Functions/Converters/DATE_TO_/Convert_DATE_TO_DATE.TcPOU
FUNCTION Convert_DATE_TO_DATE : Hresult
VAR_INPUT
	in : DATE;
	out : REFERENCE TO DATE;
END_VAR

out := in;

END_FUNCTION

// ---- Functions/Converters/DATE_TO_/Convert_DATE_TO_DINT.TcPOU
FUNCTION Convert_DATE_TO_DINT : Hresult
VAR_INPUT
	in : DATE;
	out : REFERENCE TO DINT;
END_VAR
VAR
	converted : DINT;
END_VAR

converted := DATE_TO_DINT(in);

IF (DINT_TO_DATE(converted) <> in) THEN
	Convert_DATE_TO_DINT := INCOMPATIBLE;
	RETURN;
END_IF

out := converted;

END_FUNCTION

// ---- Functions/Converters/DATE_TO_/Convert_DATE_TO_INT.TcPOU
FUNCTION Convert_DATE_TO_INT : Hresult
VAR_INPUT
	in : DATE;
	out : REFERENCE TO INT;
END_VAR
VAR
	converted : INT;
END_VAR

converted := DATE_TO_INT(in);

IF (INT_TO_DATE(converted) <> in) THEN
	Convert_DATE_TO_INT := INCOMPATIBLE;
	RETURN;
END_IF

out := converted;

END_FUNCTION

// ---- Functions/Converters/DATE_TO_/Convert_DATE_TO_REAL.TcPOU
FUNCTION Convert_DATE_TO_REAL : Hresult
VAR_INPUT
	in : DATE;
	out : REFERENCE TO REAL;
END_VAR
VAR
	converted : REAL;
END_VAR

converted := DATE_TO_REAL(in);

IF (REAL_TO_DATE(converted) <> in) THEN
	Convert_DATE_TO_REAL := INCOMPATIBLE;
	RETURN;
END_IF

out := converted;

END_FUNCTION

// ---- Functions/Converters/DATE_TO_/Convert_DATE_TO_SINT.TcPOU
FUNCTION Convert_DATE_TO_SINT : Hresult
VAR_INPUT
	in : DATE;
	out : REFERENCE TO SINT;
END_VAR
VAR
	converted : SINT;
END_VAR

converted := DATE_TO_SINT(in);

IF (SINT_TO_DATE(converted) <> in) THEN
	Convert_DATE_TO_SINT := INCOMPATIBLE;
	RETURN;
END_IF

out := converted;

END_FUNCTION

// ---- Functions/Converters/DATE_TO_/Convert_DATE_TO_STRING.TcPOU
FUNCTION Convert_DATE_TO_STRING : Hresult
VAR_INPUT
	in : DATE;
	out : REFERENCE TO STRING;
END_VAR
VAR
	converted : STRING;
END_VAR

converted := DATE_TO_STRING(in);

IF (STRING_TO_DATE(converted) <> in) THEN
	Convert_DATE_TO_STRING := INCOMPATIBLE;
	RETURN;
END_IF

out := converted;

END_FUNCTION

// ---- Functions/Converters/DATE_TO_/Convert_DATE_TO_TIME.TcPOU
FUNCTION Convert_DATE_TO_TIME : Hresult
VAR_INPUT
	in : DATE;
	out : REFERENCE TO TIME;
END_VAR
VAR
	converted : TIME;
END_VAR

converted := DATE_TO_TIME(in);

IF (TIME_TO_DATE(converted) <> in) THEN
	Convert_DATE_TO_TIME := INCOMPATIBLE;
	RETURN;
END_IF

out := converted;

END_FUNCTION

// ---- Functions/Converters/DATE_TO_/Convert_DATE_TO_TOD.TcPOU
FUNCTION Convert_DATE_TO_TOD : Hresult
VAR_INPUT
	in : DATE;
	out : REFERENCE TO TOD;
END_VAR
VAR
	converted : TOD;
END_VAR

converted := DATE_TO_TOD(in);

IF (TOD_TO_DATE(converted) <> in) THEN
	Convert_DATE_TO_TOD := INCOMPATIBLE;
	RETURN;
END_IF

out := converted;

END_FUNCTION

// ---- Functions/Converters/DATE_TO_/Convert_DATE_TO_UDINT.TcPOU
FUNCTION Convert_DATE_TO_UDINT : Hresult
VAR_INPUT
	in : DATE;
	out : REFERENCE TO UDINT;
END_VAR
VAR
	converted : UDINT;
END_VAR

converted := DATE_TO_UDINT(in);

IF (UDINT_TO_DATE(converted) <> in) THEN
	Convert_DATE_TO_UDINT := INCOMPATIBLE;
	RETURN;
END_IF

out := converted;

END_FUNCTION

// ---- Functions/Converters/DATE_TO_/Convert_DATE_TO_WORD.TcPOU
FUNCTION Convert_DATE_TO_WORD : Hresult
VAR_INPUT
	in : DATE;
	out : REFERENCE TO WORD;
END_VAR
VAR
	converted : WORD;
END_VAR

converted := DATE_TO_WORD(in);

IF (WORD_TO_DATE(converted) <> in) THEN
	Convert_DATE_TO_WORD := INCOMPATIBLE;
	RETURN;
END_IF

out := converted;

END_FUNCTION

// ---- Functions/Converters/DINT_TO_/Convert_DINT_TO_.TcPOU
FUNCTION Convert_DINT_TO_ : Hresult
VAR_INPUT
	in : DINT;
	out : ANY;
END_VAR
VAR
	convertResult : HRESULT := INCOMPATIBLE;
	convertAddress : PVOID;
	_BOOL : BOOL;
	_BYTE : BYTE;
	_DATE : DATE;
	_DINT : DINT;
	_DT : DT;
	_DWORD : DWORD;
	_INT : INT;
	_LINT : LINT;
	_LREAL : LREAL;
	_LWORD : LWORD;
	_REAL : REAL;
	_SINT : SINT;
	_STRING : STRING;
	_TIME : TIME;
	_TOD : TOD;
	_UDINT : UDINT;
	_UINT : UINT;
	_ULINT : ULINT;
	_USINT : USINT;
	_WORD : WORD;
END_VAR

CASE out.TypeClass OF
	
	__SYSTEM.TYPE_CLASS.TYPE_BOOL:
	
		convertResult := Convert_DINT_TO_BOOL(in, _BOOL);
		IF SUCCEEDED(convertResult) THEN
			convertAddress := ADR(_BOOL);
		END_IF

	__SYSTEM.TYPE_CLASS.TYPE_BYTE:
	
		convertResult := Convert_DINT_TO_BYTE(in, _BYTE);
		IF SUCCEEDED(convertResult) THEN
			convertAddress := ADR(_BYTE);
		END_IF

	__SYSTEM.TYPE_CLASS.TYPE_DATE:
	
		convertResult := Convert_DINT_TO_DATE(in, _DATE);
		IF SUCCEEDED(convertResult) THEN
			convertAddress := ADR(_DATE);
		END_IF

	__SYSTEM.TYPE_CLASS.TYPE_DINT:
	
		convertResult := Convert_DINT_TO_DINT(in, _DINT);
		IF SUCCEEDED(convertResult) THEN
			convertAddress := ADR(_DINT);
		END_IF

	__SYSTEM.TYPE_CLASS.TYPE_DATEANDTIME:
	
		convertResult := Convert_DINT_TO_DT(in, _DT);
		IF SUCCEEDED(convertResult) THEN
			convertAddress := ADR(_DT);
		END_IF

	__SYSTEM.TYPE_CLASS.TYPE_DWORD:
	
		convertResult := Convert_DINT_TO_DWORD(in, _DWORD);
		IF SUCCEEDED(convertResult) THEN
			convertAddress := ADR(_DWORD);
		END_IF

	__SYSTEM.TYPE_CLASS.TYPE_INT:
	
		convertResult := Convert_DINT_TO_INT(in, _INT);
		IF SUCCEEDED(convertResult) THEN
			convertAddress := ADR(_INT);
		END_IF

	__SYSTEM.TYPE_CLASS.TYPE_LINT:
	
		convertResult := Convert_DINT_TO_LINT(in, _LINT);
		IF SUCCEEDED(convertResult) THEN
			convertAddress := ADR(_LINT);
		END_IF

	__SYSTEM.TYPE_CLASS.TYPE_LREAL:
	
		convertResult := Convert_DINT_TO_LREAL(in, _LREAL);
		IF SUCCEEDED(convertResult) THEN
			convertAddress := ADR(_LREAL);
		END_IF

	__SYSTEM.TYPE_CLASS.TYPE_LWORD:
	
		convertResult := Convert_DINT_TO_LWORD(in, _LWORD);
		IF SUCCEEDED(convertResult) THEN
			convertAddress := ADR(_LWORD);
		END_IF

	__SYSTEM.TYPE_CLASS.TYPE_REAL:
	
		convertResult := Convert_DINT_TO_REAL(in, _REAL);
		IF SUCCEEDED(convertResult) THEN
			convertAddress := ADR(_REAL);
		END_IF

	__SYSTEM.TYPE_CLASS.TYPE_SINT:
	
		convertResult := Convert_DINT_TO_SINT(in, _SINT);
		IF SUCCEEDED(convertResult) THEN
			convertAddress := ADR(_SINT);
		END_IF

	__SYSTEM.TYPE_CLASS.TYPE_STRING:
	
		convertResult := Convert_DINT_TO_STRING(in, _STRING);
		IF SUCCEEDED(convertResult) THEN
			convertAddress := ADR(_STRING);
		END_IF

	__SYSTEM.TYPE_CLASS.TYPE_TIME:
	
		convertResult := Convert_DINT_TO_TIME(in, _TIME);
		IF SUCCEEDED(convertResult) THEN
			convertAddress := ADR(_TIME);
		END_IF

	__SYSTEM.TYPE_CLASS.TYPE_TIMEOFDAY:
	
		convertResult := Convert_DINT_TO_TOD(in, _TOD);
		IF SUCCEEDED(convertResult) THEN
			convertAddress := ADR(_TOD);
		END_IF

	__SYSTEM.TYPE_CLASS.TYPE_UDINT:
	
		convertResult := Convert_DINT_TO_UDINT(in, _UDINT);
		IF SUCCEEDED(convertResult) THEN
			convertAddress := ADR(_UDINT);
		END_IF

	__SYSTEM.TYPE_CLASS.TYPE_UINT:
	
		convertResult := Convert_DINT_TO_UINT(in, _UINT);
		IF SUCCEEDED(convertResult) THEN
			convertAddress := ADR(_UINT);
		END_IF

	__SYSTEM.TYPE_CLASS.TYPE_ULINT:
	
		convertResult := Convert_DINT_TO_ULINT(in, _ULINT);
		IF SUCCEEDED(convertResult) THEN
			convertAddress := ADR(_ULINT);
		END_IF

	__SYSTEM.TYPE_CLASS.TYPE_USINT:
	
		convertResult := Convert_DINT_TO_USINT(in, _USINT);
		IF SUCCEEDED(convertResult) THEN
			convertAddress := ADR(_USINT);
		END_IF

	__SYSTEM.TYPE_CLASS.TYPE_WORD:
	
		convertResult := Convert_DINT_TO_WORD(in, _WORD);
		IF SUCCEEDED(convertResult) THEN
			convertAddress := ADR(_WORD);
		END_IF

END_CASE

IF SUCCEEDED(convertResult) THEN
	memcpy(out.pValue,convertAddress,DINT_TO_UDINT(out.diSize));
END_IF

Convert_DINT_TO_ := convertResult;

END_FUNCTION

// ---- Functions/Converters/DINT_TO_/Convert_DINT_TO_BOOL.TcPOU
FUNCTION Convert_DINT_TO_BOOL : Hresult
VAR_INPUT
	in : DINT;
	out : REFERENCE TO BOOL;
END_VAR
VAR
	converted : BOOL;
END_VAR

converted := DINT_TO_BOOL(in);

IF (BOOL_TO_DINT(converted) <> in) THEN
	Convert_DINT_TO_BOOL := INCOMPATIBLE;
	RETURN;
END_IF

out := converted;

END_FUNCTION

// ---- Functions/Converters/DINT_TO_/Convert_DINT_TO_BYTE.TcPOU
FUNCTION Convert_DINT_TO_BYTE : Hresult
VAR_INPUT
	in : DINT;
	out : REFERENCE TO BYTE;
END_VAR
VAR
	converted : BYTE;
END_VAR

converted := DINT_TO_BYTE(in);

IF (BYTE_TO_DINT(converted) <> in) THEN
	Convert_DINT_TO_BYTE := INCOMPATIBLE;
	RETURN;
END_IF

out := converted;

END_FUNCTION

// ---- Functions/Converters/DINT_TO_/Convert_DINT_TO_DWORD.TcPOU
FUNCTION Convert_DINT_TO_DWORD : Hresult
VAR_INPUT
	in : DINT;
	out : REFERENCE TO DWORD;
END_VAR
VAR
	converted : DWORD;
END_VAR

converted := DINT_TO_DWORD(in);

IF (DWORD_TO_DINT(converted) <> in) THEN
	Convert_DINT_TO_DWORD := INCOMPATIBLE;
	RETURN;
END_IF

out := converted;

END_FUNCTION

// ---- Functions/Converters/DINT_TO_/Convert_DINT_TO_INT.TcPOU
FUNCTION Convert_DINT_TO_INT : Hresult
VAR_INPUT
	in : DINT;
	out : REFERENCE TO INT;
END_VAR
VAR
	converted : INT;
END_VAR

converted := DINT_TO_INT(in);

IF (INT_TO_DINT(converted) <> in) THEN
	Convert_DINT_TO_INT := INCOMPATIBLE;
	RETURN;
END_IF

out := converted;

END_FUNCTION

// ---- Functions/Converters/DINT_TO_/Convert_DINT_TO_LINT.TcPOU
FUNCTION Convert_DINT_TO_LINT : Hresult
VAR_INPUT
	in : DINT;
	out : REFERENCE TO LINT;
END_VAR
VAR
	converted : LINT;
END_VAR

converted := DINT_TO_LINT(in);

IF (LINT_TO_DINT(converted) <> in) THEN
	Convert_DINT_TO_LINT := INCOMPATIBLE;
	RETURN;
END_IF

out := converted;

END_FUNCTION

// ---- Functions/Converters/DINT_TO_/Convert_DINT_TO_LWORD.TcPOU
FUNCTION Convert_DINT_TO_LWORD : Hresult
VAR_INPUT
	in : DINT;
	out : REFERENCE TO LWORD;
END_VAR
VAR
	converted : LWORD;
END_VAR

converted := DINT_TO_LWORD(in);

IF (LWORD_TO_DINT(converted) <> in) THEN
	Convert_DINT_TO_LWORD := INCOMPATIBLE;
	RETURN;
END_IF

out := converted;

END_FUNCTION

// ---- Functions/Converters/DINT_TO_/Convert_DINT_TO_SINT.TcPOU
FUNCTION Convert_DINT_TO_SINT : Hresult
VAR_INPUT
	in : DINT;
	out : REFERENCE TO SINT;
END_VAR
VAR
	converted : SINT;
END_VAR

converted := DINT_TO_SINT(in);

IF (SINT_TO_DINT(converted) <> in) THEN
	Convert_DINT_TO_SINT := INCOMPATIBLE;
	RETURN;
END_IF

out := converted;

END_FUNCTION

// ---- Functions/Converters/DINT_TO_/Convert_DINT_TO_STRING.TcPOU
FUNCTION Convert_DINT_TO_STRING : Hresult
VAR_INPUT
	in : DINT;
	out : REFERENCE TO STRING;
END_VAR
VAR
	converted : STRING;
END_VAR

converted := DINT_TO_STRING(in);

IF (STRING_TO_DINT(converted) <> in) THEN
	Convert_DINT_TO_STRING := INCOMPATIBLE;
	RETURN;
END_IF

out := converted;

END_FUNCTION

// ---- Functions/Converters/DINT_TO_/Convert_DINT_TO_UDINT.TcPOU
FUNCTION Convert_DINT_TO_UDINT : Hresult
VAR_INPUT
	in : DINT;
	out : REFERENCE TO UDINT;
END_VAR
VAR
	converted : UDINT;
END_VAR

converted := DINT_TO_UDINT(in);

IF (UDINT_TO_DINT(converted) <> in) THEN
	Convert_DINT_TO_UDINT := INCOMPATIBLE;
	RETURN;
END_IF

out := converted;

END_FUNCTION

// ---- Functions/Converters/DINT_TO_/Convert_DINT_TO_USINT.TcPOU
FUNCTION Convert_DINT_TO_USINT : Hresult
VAR_INPUT
	in : DINT;
	out : REFERENCE TO USINT;
END_VAR
VAR
	converted : USINT;
END_VAR

converted := DINT_TO_USINT(in);

IF (USINT_TO_DINT(converted) <> in) THEN
	Convert_DINT_TO_USINT := INCOMPATIBLE;
	RETURN;
END_IF

out := converted;

END_FUNCTION

// ---- Functions/Converters/DINT_TO_/Convert_DINT_TO_WORD.TcPOU
FUNCTION Convert_DINT_TO_WORD : Hresult
VAR_INPUT
	in : DINT;
	out : REFERENCE TO WORD;
END_VAR
VAR
	converted : WORD;
END_VAR

converted := DINT_TO_WORD(in);

IF (WORD_TO_DINT(converted) <> in) THEN
	Convert_DINT_TO_WORD := INCOMPATIBLE;
	RETURN;
END_IF

out := converted;

END_FUNCTION

// ---- Functions/Converters/DT_TO_/Convert_DT_TO_BOOL.TcPOU
FUNCTION Convert_DT_TO_BOOL : Hresult
VAR_INPUT
	in : DT;
	out : REFERENCE TO BOOL;
END_VAR
VAR
	converted : BOOL;
END_VAR

converted := DT_TO_BOOL(in);

IF (BOOL_TO_DT(converted) <> in) THEN
	Convert_DT_TO_BOOL := INCOMPATIBLE;
	RETURN;
END_IF

out := converted;

END_FUNCTION

// ---- Functions/Converters/DT_TO_/Convert_DT_TO_BYTE.TcPOU
FUNCTION Convert_DT_TO_BYTE : Hresult
VAR_INPUT
	in : DT;
	out : REFERENCE TO BYTE;
END_VAR
VAR
	converted : BYTE;
END_VAR

converted := DT_TO_BYTE(in);

IF (BYTE_TO_DT(converted) <> in) THEN
	Convert_DT_TO_BYTE := INCOMPATIBLE;
	RETURN;
END_IF

out := converted;

END_FUNCTION

// ---- Functions/Converters/DT_TO_/Convert_DT_TO_DATE.TcPOU
FUNCTION Convert_DT_TO_DATE : Hresult
VAR_INPUT
	in : DT;
	out : REFERENCE TO DATE;
END_VAR
VAR
	converted : DATE;
END_VAR

converted := DT_TO_DATE(in);

IF (DATE_TO_DT(converted) <> in) THEN
	Convert_DT_TO_DATE := INCOMPATIBLE;
	RETURN;
END_IF

out := converted;

END_FUNCTION

// ---- Functions/Converters/DT_TO_/Convert_DT_TO_DWORD.TcPOU
FUNCTION Convert_DT_TO_DWORD : Hresult
VAR_INPUT
	in : DT;
	out : REFERENCE TO DWORD;
END_VAR
VAR
	converted : DWORD;
END_VAR

converted := DT_TO_DWORD(in);

IF (DWORD_TO_DT(converted) <> in) THEN
	Convert_DT_TO_DWORD := INCOMPATIBLE;
	RETURN;
END_IF

out := converted;

END_FUNCTION

// ---- Functions/Converters/DT_TO_/Convert_DT_TO_INT.TcPOU
FUNCTION Convert_DT_TO_INT : Hresult
VAR_INPUT
	in : DT;
	out : REFERENCE TO INT;
END_VAR
VAR
	converted : INT;
END_VAR

converted := DT_TO_INT(in);

IF (INT_TO_DT(converted) <> in) THEN
	Convert_DT_TO_INT := INCOMPATIBLE;
	RETURN;
END_IF

out := converted;

END_FUNCTION

// ---- Functions/Converters/DT_TO_/Convert_DT_TO_LWORD.TcPOU
FUNCTION Convert_DT_TO_LWORD : Hresult
VAR_INPUT
	in : DT;
	out : REFERENCE TO LWORD;
END_VAR
VAR
	converted : LWORD;
END_VAR

converted := DT_TO_LWORD(in);

IF (LWORD_TO_DT(converted) <> in) THEN
	Convert_DT_TO_LWORD := INCOMPATIBLE;
	RETURN;
END_IF

out := converted;

END_FUNCTION

// ---- Functions/Converters/DT_TO_/Convert_DT_TO_REAL.TcPOU
FUNCTION Convert_DT_TO_REAL : Hresult
VAR_INPUT
	in : DT;
	out : REFERENCE TO REAL;
END_VAR
VAR
	converted : REAL;
END_VAR

converted := DT_TO_REAL(in);

IF (REAL_TO_DT(converted) <> in) THEN
	Convert_DT_TO_REAL := INCOMPATIBLE;
	RETURN;
END_IF

out := converted;

END_FUNCTION

// ---- Functions/Converters/DT_TO_/Convert_DT_TO_SINT.TcPOU
FUNCTION Convert_DT_TO_SINT : Hresult
VAR_INPUT
	in : DT;
	out : REFERENCE TO SINT;
END_VAR
VAR
	converted : SINT;
END_VAR

converted := DT_TO_SINT(in);

IF (SINT_TO_DT(converted) <> in) THEN
	Convert_DT_TO_SINT := INCOMPATIBLE;
	RETURN;
END_IF

out := converted;

END_FUNCTION

// ---- Functions/Converters/DT_TO_/Convert_DT_TO_STRING.TcPOU
FUNCTION Convert_DT_TO_STRING : Hresult
VAR_INPUT
	in : DT;
	out : REFERENCE TO STRING;
END_VAR
VAR
	converted : STRING;
END_VAR

converted := DT_TO_STRING(in);

IF (STRING_TO_DT(converted) <> in) THEN
	Convert_DT_TO_STRING := INCOMPATIBLE;
	RETURN;
END_IF

out := converted;

END_FUNCTION

// ---- Functions/Converters/DT_TO_/Convert_DT_TO_UDINT.TcPOU
FUNCTION Convert_DT_TO_UDINT : Hresult
VAR_INPUT
	in : DT;
	out : REFERENCE TO UDINT;
END_VAR
VAR
	converted : UDINT;
END_VAR

converted := DT_TO_UDINT(in);

IF (UDINT_TO_DT(converted) <> in) THEN
	Convert_DT_TO_UDINT := INCOMPATIBLE;
	RETURN;
END_IF

out := converted;

END_FUNCTION

// ---- Functions/Converters/DT_TO_/Convert_DT_TO_UINT.TcPOU
FUNCTION Convert_DT_TO_UINT : Hresult
VAR_INPUT
	in : DT;
	out : REFERENCE TO UINT;
END_VAR
VAR
	converted : UINT;
END_VAR

converted := DT_TO_UINT(in);

IF (UINT_TO_DT(converted) <> in) THEN
	Convert_DT_TO_UINT := INCOMPATIBLE;
	RETURN;
END_IF

out := converted;

END_FUNCTION

// ---- Functions/Converters/DT_TO_/Convert_DT_TO_USINT.TcPOU
FUNCTION Convert_DT_TO_USINT : Hresult
VAR_INPUT
	in : DT;
	out : REFERENCE TO USINT;
END_VAR
VAR
	converted : USINT;
END_VAR

converted := DT_TO_USINT(in);

IF (USINT_TO_DT(converted) <> in) THEN
	Convert_DT_TO_USINT := INCOMPATIBLE;
	RETURN;
END_IF

out := converted;

END_FUNCTION

// ---- Functions/Converters/DWORD_TO_/Convert_DWORD_TO_.TcPOU
FUNCTION Convert_DWORD_TO_ : Hresult
VAR_INPUT
	in : DWORD;
	out : ANY;
END_VAR
VAR
	convertResult : HRESULT := INCOMPATIBLE;
	convertAddress : PVOID;
	_BOOL : BOOL;
	_BYTE : BYTE;
	_DATE : DATE;
	_DINT : DINT;
	_DT : DT;
	_DWORD : DWORD;
	_INT : INT;
	_LINT : LINT;
	_LREAL : LREAL;
	_LWORD : LWORD;
	_REAL : REAL;
	_SINT : SINT;
	_STRING : STRING;
	_TIME : TIME;
	_TOD : TOD;
	_UDINT : UDINT;
	_UINT : UINT;
	_ULINT : ULINT;
	_USINT : USINT;
	_WORD : WORD;
END_VAR

CASE out.TypeClass OF
	
	__SYSTEM.TYPE_CLASS.TYPE_BOOL:
	
		convertResult := Convert_DWORD_TO_BOOL(in, _BOOL);
		IF SUCCEEDED(convertResult) THEN
			convertAddress := ADR(_BOOL);
		END_IF

	__SYSTEM.TYPE_CLASS.TYPE_BYTE:
	
		convertResult := Convert_DWORD_TO_BYTE(in, _BYTE);
		IF SUCCEEDED(convertResult) THEN
			convertAddress := ADR(_BYTE);
		END_IF

	__SYSTEM.TYPE_CLASS.TYPE_DATE:
	
		convertResult := Convert_DWORD_TO_DATE(in, _DATE);
		IF SUCCEEDED(convertResult) THEN
			convertAddress := ADR(_DATE);
		END_IF

	__SYSTEM.TYPE_CLASS.TYPE_DINT:
	
		convertResult := Convert_DWORD_TO_DINT(in, _DINT);
		IF SUCCEEDED(convertResult) THEN
			convertAddress := ADR(_DINT);
		END_IF

	__SYSTEM.TYPE_CLASS.TYPE_DATEANDTIME:
	
		convertResult := Convert_DWORD_TO_DT(in, _DT);
		IF SUCCEEDED(convertResult) THEN
			convertAddress := ADR(_DT);
		END_IF

	__SYSTEM.TYPE_CLASS.TYPE_DWORD:
	
		convertResult := Convert_DWORD_TO_DWORD(in, _DWORD);
		IF SUCCEEDED(convertResult) THEN
			convertAddress := ADR(_DWORD);
		END_IF

	__SYSTEM.TYPE_CLASS.TYPE_INT:
	
		convertResult := Convert_DWORD_TO_INT(in, _INT);
		IF SUCCEEDED(convertResult) THEN
			convertAddress := ADR(_INT);
		END_IF

	__SYSTEM.TYPE_CLASS.TYPE_LINT:
	
		convertResult := Convert_DWORD_TO_LINT(in, _LINT);
		IF SUCCEEDED(convertResult) THEN
			convertAddress := ADR(_LINT);
		END_IF

	__SYSTEM.TYPE_CLASS.TYPE_LREAL:
	
		convertResult := Convert_DWORD_TO_LREAL(in, _LREAL);
		IF SUCCEEDED(convertResult) THEN
			convertAddress := ADR(_LREAL);
		END_IF

	__SYSTEM.TYPE_CLASS.TYPE_LWORD:
	
		convertResult := Convert_DWORD_TO_LWORD(in, _LWORD);
		IF SUCCEEDED(convertResult) THEN
			convertAddress := ADR(_LWORD);
		END_IF

	__SYSTEM.TYPE_CLASS.TYPE_REAL:
	
		convertResult := Convert_DWORD_TO_REAL(in, _REAL);
		IF SUCCEEDED(convertResult) THEN
			convertAddress := ADR(_REAL);
		END_IF

	__SYSTEM.TYPE_CLASS.TYPE_SINT:
	
		convertResult := Convert_DWORD_TO_SINT(in, _SINT);
		IF SUCCEEDED(convertResult) THEN
			convertAddress := ADR(_SINT);
		END_IF

	__SYSTEM.TYPE_CLASS.TYPE_STRING:
	
		convertResult := Convert_DWORD_TO_STRING(in, _STRING);
		IF SUCCEEDED(convertResult) THEN
			convertAddress := ADR(_STRING);
		END_IF

	__SYSTEM.TYPE_CLASS.TYPE_TIME:
	
		convertResult := Convert_DWORD_TO_TIME(in, _TIME);
		IF SUCCEEDED(convertResult) THEN
			convertAddress := ADR(_TIME);
		END_IF

	__SYSTEM.TYPE_CLASS.TYPE_TIMEOFDAY:
	
		convertResult := Convert_DWORD_TO_TOD(in, _TOD);
		IF SUCCEEDED(convertResult) THEN
			convertAddress := ADR(_TOD);
		END_IF

	__SYSTEM.TYPE_CLASS.TYPE_UDINT:
	
		convertResult := Convert_DWORD_TO_UDINT(in, _UDINT);
		IF SUCCEEDED(convertResult) THEN
			convertAddress := ADR(_UDINT);
		END_IF

	__SYSTEM.TYPE_CLASS.TYPE_UINT:
	
		convertResult := Convert_DWORD_TO_UINT(in, _UINT);
		IF SUCCEEDED(convertResult) THEN
			convertAddress := ADR(_UINT);
		END_IF

	__SYSTEM.TYPE_CLASS.TYPE_ULINT:
	
		convertResult := Convert_DWORD_TO_ULINT(in, _ULINT);
		IF SUCCEEDED(convertResult) THEN
			convertAddress := ADR(_ULINT);
		END_IF

	__SYSTEM.TYPE_CLASS.TYPE_USINT:
	
		convertResult := Convert_DWORD_TO_USINT(in, _USINT);
		IF SUCCEEDED(convertResult) THEN
			convertAddress := ADR(_USINT);
		END_IF

	__SYSTEM.TYPE_CLASS.TYPE_WORD:
	
		convertResult := Convert_DWORD_TO_WORD(in, _WORD);
		IF SUCCEEDED(convertResult) THEN
			convertAddress := ADR(_WORD);
		END_IF

END_CASE

IF SUCCEEDED(convertResult) THEN
	memcpy(out.pValue,convertAddress,DINT_TO_UDINT(out.diSize));
END_IF

Convert_DWORD_TO_ := convertResult;

END_FUNCTION

// ---- Functions/Converters/DWORD_TO_/Convert_DWORD_TO_BYTE.TcPOU
FUNCTION Convert_DWORD_TO_BYTE : Hresult
VAR_INPUT
	in : DWORD;
	out : REFERENCE TO BYTE;
END_VAR
VAR
	converted : BYTE;
END_VAR

converted := DWORD_TO_BYTE(in);

IF (BYTE_TO_DWORD(converted) <> in) THEN
	Convert_DWORD_TO_BYTE := INCOMPATIBLE;
	RETURN;
END_IF

out := converted;

END_FUNCTION

// ---- Functions/Converters/DWORD_TO_/Convert_DWORD_TO_DATE.TcPOU
FUNCTION Convert_DWORD_TO_DATE : Hresult
VAR_INPUT
	in : DWORD;
	out : REFERENCE TO DATE;
END_VAR
VAR
	converted : DATE;
END_VAR

converted := DWORD_TO_DATE(in);

IF (DATE_TO_DWORD(converted) <> in) THEN
	Convert_DWORD_TO_DATE := INCOMPATIBLE;
	RETURN;
END_IF

out := converted;

END_FUNCTION

// ---- Functions/Converters/DWORD_TO_/Convert_DWORD_TO_DWORD.TcPOU
FUNCTION Convert_DWORD_TO_DWORD : Hresult
VAR_INPUT
	in : DWORD;
	out : REFERENCE TO DWORD;
END_VAR

out := in;

END_FUNCTION

// ---- Functions/Converters/DWORD_TO_/Convert_DWORD_TO_INT.TcPOU
FUNCTION Convert_DWORD_TO_INT : Hresult
VAR_INPUT
	in : DWORD;
	out : REFERENCE TO INT;
END_VAR
VAR
	converted : INT;
END_VAR

converted := DWORD_TO_INT(in);

IF (INT_TO_DWORD(converted) <> in) THEN
	Convert_DWORD_TO_INT := INCOMPATIBLE;
	RETURN;
END_IF

out := converted;

END_FUNCTION

// ---- Functions/Converters/DWORD_TO_/Convert_DWORD_TO_LINT.TcPOU
FUNCTION Convert_DWORD_TO_LINT : Hresult
VAR_INPUT
	in : DWORD;
	out : REFERENCE TO LINT;
END_VAR
VAR
	converted : LINT;
END_VAR

converted := DWORD_TO_LINT(in);

IF (LINT_TO_DWORD(converted) <> in) THEN
	Convert_DWORD_TO_LINT := INCOMPATIBLE;
	RETURN;
END_IF

out := converted;

END_FUNCTION

// ---- Functions/Converters/DWORD_TO_/Convert_DWORD_TO_LWORD.TcPOU
FUNCTION Convert_DWORD_TO_LWORD : Hresult
VAR_INPUT
	in : DWORD;
	out : REFERENCE TO LWORD;
END_VAR
VAR
	converted : LWORD;
END_VAR

converted := DWORD_TO_LWORD(in);

IF (LWORD_TO_DWORD(converted) <> in) THEN
	Convert_DWORD_TO_LWORD := INCOMPATIBLE;
	RETURN;
END_IF

out := converted;

END_FUNCTION

// ---- Functions/Converters/DWORD_TO_/Convert_DWORD_TO_REAL.TcPOU
FUNCTION Convert_DWORD_TO_REAL : Hresult
VAR_INPUT
	in : DWORD;
	out : REFERENCE TO REAL;
END_VAR
VAR
	converted : REAL;
END_VAR

converted := DWORD_TO_REAL(in);

IF (REAL_TO_DWORD(converted) <> in) THEN
	Convert_DWORD_TO_REAL := INCOMPATIBLE;
	RETURN;
END_IF

out := converted;

END_FUNCTION

// ---- Functions/Converters/DWORD_TO_/Convert_DWORD_TO_TOD.TcPOU
FUNCTION Convert_DWORD_TO_TOD : Hresult
VAR_INPUT
	in : DWORD;
	out : REFERENCE TO TOD;
END_VAR
VAR
	converted : TOD;
END_VAR

converted := DWORD_TO_TOD(in);

IF (TOD_TO_DWORD(converted) <> in) THEN
	Convert_DWORD_TO_TOD := INCOMPATIBLE;
	RETURN;
END_IF

out := converted;

END_FUNCTION

// ---- Functions/Converters/DWORD_TO_/Convert_DWORD_TO_UDINT.TcPOU
FUNCTION Convert_DWORD_TO_UDINT : Hresult
VAR_INPUT
	in : DWORD;
	out : REFERENCE TO UDINT;
END_VAR
VAR
	converted : UDINT;
END_VAR

converted := DWORD_TO_UDINT(in);

IF (UDINT_TO_DWORD(converted) <> in) THEN
	Convert_DWORD_TO_UDINT := INCOMPATIBLE;
	RETURN;
END_IF

out := converted;

END_FUNCTION

// ---- Functions/Converters/DWORD_TO_/Convert_DWORD_TO_UINT.TcPOU
FUNCTION Convert_DWORD_TO_UINT : Hresult
VAR_INPUT
	in : DWORD;
	out : REFERENCE TO UINT;
END_VAR
VAR
	converted : UINT;
END_VAR

converted := DWORD_TO_UINT(in);

IF (UINT_TO_DWORD(converted) <> in) THEN
	Convert_DWORD_TO_UINT := INCOMPATIBLE;
	RETURN;
END_IF

out := converted;

END_FUNCTION

// ---- Functions/Converters/DWORD_TO_/Convert_DWORD_TO_ULINT.TcPOU
FUNCTION Convert_DWORD_TO_ULINT : Hresult
VAR_INPUT
	in : DWORD;
	out : REFERENCE TO ULINT;
END_VAR
VAR
	converted : ULINT;
END_VAR

converted := DWORD_TO_ULINT(in);

IF (ULINT_TO_DWORD(converted) <> in) THEN
	Convert_DWORD_TO_ULINT := INCOMPATIBLE;
	RETURN;
END_IF

out := converted;

END_FUNCTION

// ---- Functions/Converters/DWORD_TO_/Convert_DWORD_TO_WORD.TcPOU
FUNCTION Convert_DWORD_TO_WORD : Hresult
VAR_INPUT
	in : DWORD;
	out : REFERENCE TO WORD;
END_VAR
VAR
	converted : WORD;
END_VAR

converted := DWORD_TO_WORD(in);

IF (WORD_TO_DWORD(converted) <> in) THEN
	Convert_DWORD_TO_WORD := INCOMPATIBLE;
	RETURN;
END_IF

out := converted;

END_FUNCTION

// ---- Functions/Converters/INT_TO_/Convert_INT_TO_BYTE.TcPOU
FUNCTION Convert_INT_TO_BYTE : Hresult
VAR_INPUT
	in : INT;
	out : REFERENCE TO BYTE;
END_VAR
VAR
	converted : BYTE;
END_VAR

converted := INT_TO_BYTE(in);

IF (BYTE_TO_INT(converted) <> in) THEN
	Convert_INT_TO_BYTE := INCOMPATIBLE;
	RETURN;
END_IF

out := converted;

END_FUNCTION

// ---- Functions/Converters/INT_TO_/Convert_INT_TO_DT.TcPOU
FUNCTION Convert_INT_TO_DT : Hresult
VAR_INPUT
	in : INT;
	out : REFERENCE TO DT;
END_VAR
VAR
	converted : DT;
END_VAR

converted := INT_TO_DT(in);

IF (DT_TO_INT(converted) <> in) THEN
	Convert_INT_TO_DT := INCOMPATIBLE;
	RETURN;
END_IF

out := converted;

END_FUNCTION

// ---- Functions/Converters/INT_TO_/Convert_INT_TO_LREAL.TcPOU
FUNCTION Convert_INT_TO_LREAL : Hresult
VAR_INPUT
	in : INT;
	out : REFERENCE TO LREAL;
END_VAR
VAR
	converted : LREAL;
END_VAR

converted := INT_TO_LREAL(in);

IF (LREAL_TO_INT(converted) <> in) THEN
	Convert_INT_TO_LREAL := INCOMPATIBLE;
	RETURN;
END_IF

out := converted;

END_FUNCTION

// ---- Functions/Converters/INT_TO_/Convert_INT_TO_LWORD.TcPOU
FUNCTION Convert_INT_TO_LWORD : Hresult
VAR_INPUT
	in : INT;
	out : REFERENCE TO LWORD;
END_VAR
VAR
	converted : LWORD;
END_VAR

converted := INT_TO_LWORD(in);

IF (LWORD_TO_INT(converted) <> in) THEN
	Convert_INT_TO_LWORD := INCOMPATIBLE;
	RETURN;
END_IF

out := converted;

END_FUNCTION

// ---- Functions/Converters/INT_TO_/Convert_INT_TO_STRING.TcPOU
FUNCTION Convert_INT_TO_STRING : Hresult
VAR_INPUT
	in : INT;
	out : REFERENCE TO STRING;
END_VAR
VAR
	converted : STRING;
END_VAR

converted := INT_TO_STRING(in);

IF (STRING_TO_INT(converted) <> in) THEN
	Convert_INT_TO_STRING := INCOMPATIBLE;
	RETURN;
END_IF

out := converted;

END_FUNCTION

// ---- Functions/Converters/INT_TO_/Convert_INT_TO_TOD.TcPOU
FUNCTION Convert_INT_TO_TOD : Hresult
VAR_INPUT
	in : INT;
	out : REFERENCE TO TOD;
END_VAR
VAR
	converted : TOD;
END_VAR

converted := INT_TO_TOD(in);

IF (TOD_TO_INT(converted) <> in) THEN
	Convert_INT_TO_TOD := INCOMPATIBLE;
	RETURN;
END_IF

out := converted;

END_FUNCTION

// ---- Functions/Converters/LINT_TO/Convert_LINT_TO_DATE.TcPOU
FUNCTION Convert_LINT_TO_DATE : Hresult
VAR_INPUT
	in : LINT;
	out : REFERENCE TO DATE;
END_VAR
VAR
	converted : DATE;
END_VAR

converted := LINT_TO_DATE(in);

IF (DATE_TO_LINT(converted) <> in) THEN
	Convert_LINT_TO_DATE := INCOMPATIBLE;
	RETURN;
END_IF

out := converted;

END_FUNCTION

// ---- Functions/Converters/LINT_TO/Convert_LINT_TO_DWORD.TcPOU
FUNCTION Convert_LINT_TO_DWORD : Hresult
VAR_INPUT
	in : LINT;
	out : REFERENCE TO DWORD;
END_VAR
VAR
	converted : DWORD;
END_VAR

converted := LINT_TO_DWORD(in);

IF (DWORD_TO_LINT(converted) <> in) THEN
	Convert_LINT_TO_DWORD := INCOMPATIBLE;
	RETURN;
END_IF

out := converted;

END_FUNCTION

// ---- Functions/Converters/LINT_TO/Convert_LINT_TO_LWORD.TcPOU
FUNCTION Convert_LINT_TO_LWORD : Hresult
VAR_INPUT
	in : LINT;
	out : REFERENCE TO LWORD;
END_VAR
VAR
	converted : LWORD;
END_VAR

converted := LINT_TO_LWORD(in);

IF (LWORD_TO_LINT(converted) <> in) THEN
	Convert_LINT_TO_LWORD := INCOMPATIBLE;
	RETURN;
END_IF

out := converted;

END_FUNCTION

// ---- Functions/Converters/LINT_TO/Convert_LINT_TO_REAL.TcPOU
FUNCTION Convert_LINT_TO_REAL : Hresult
VAR_INPUT
	in : LINT;
	out : REFERENCE TO REAL;
END_VAR
VAR
	converted : REAL;
END_VAR

converted := LINT_TO_REAL(in);

IF (REAL_TO_LINT(converted) <> in) THEN
	Convert_LINT_TO_REAL := INCOMPATIBLE;
	RETURN;
END_IF

out := converted;

END_FUNCTION

// ---- Functions/Converters/LINT_TO/Convert_LINT_TO_SINT.TcPOU
FUNCTION Convert_LINT_TO_SINT : Hresult
VAR_INPUT
	in : LINT;
	out : REFERENCE TO SINT;
END_VAR
VAR
	converted : SINT;
END_VAR

converted := LINT_TO_SINT(in);

IF (SINT_TO_LINT(converted) <> in) THEN
	Convert_LINT_TO_SINT := INCOMPATIBLE;
	RETURN;
END_IF

out := converted;

END_FUNCTION

// ---- Functions/Converters/LINT_TO/Convert_LINT_TO_TIME.TcPOU
FUNCTION Convert_LINT_TO_TIME : Hresult
VAR_INPUT
	in : LINT;
	out : REFERENCE TO TIME;
END_VAR
VAR
	converted : TIME;
END_VAR

converted := LINT_TO_TIME(in);

IF (TIME_TO_LINT(converted) <> in) THEN
	Convert_LINT_TO_TIME := INCOMPATIBLE;
	RETURN;
END_IF

out := converted;

END_FUNCTION

// ---- Functions/Converters/LINT_TO/Convert_LINT_TO_UDINT.TcPOU
FUNCTION Convert_LINT_TO_UDINT : Hresult
VAR_INPUT
	in : LINT;
	out : REFERENCE TO UDINT;
END_VAR
VAR
	converted : UDINT;
END_VAR

converted := LINT_TO_UDINT(in);

IF (UDINT_TO_LINT(converted) <> in) THEN
	Convert_LINT_TO_UDINT := INCOMPATIBLE;
	RETURN;
END_IF

out := converted;

END_FUNCTION

// ---- Functions/Converters/LINT_TO/Convert_LINT_TO_UINT.TcPOU
FUNCTION Convert_LINT_TO_UINT : Hresult
VAR_INPUT
	in : LINT;
	out : REFERENCE TO UINT;
END_VAR
VAR
	converted : UINT;
END_VAR

converted := LINT_TO_UINT(in);

IF (UINT_TO_LINT(converted) <> in) THEN
	Convert_LINT_TO_UINT := INCOMPATIBLE;
	RETURN;
END_IF

out := converted;

END_FUNCTION

// ---- Functions/Converters/LINT_TO/Convert_LINT_TO_ULINT.TcPOU
FUNCTION Convert_LINT_TO_ULINT : Hresult
VAR_INPUT
	in : LINT;
	out : REFERENCE TO ULINT;
END_VAR
VAR
	converted : ULINT;
END_VAR

converted := LINT_TO_ULINT(in);

IF (ULINT_TO_LINT(converted) <> in) THEN
	Convert_LINT_TO_ULINT := INCOMPATIBLE;
	RETURN;
END_IF

out := converted;

END_FUNCTION

// ---- Functions/Converters/LINT_TO/Convert_LINT_TO_WORD.TcPOU
FUNCTION Convert_LINT_TO_WORD : Hresult
VAR_INPUT
	in : LINT;
	out : REFERENCE TO WORD;
END_VAR
VAR
	converted : WORD;
END_VAR

converted := LINT_TO_WORD(in);

IF (WORD_TO_LINT(converted) <> in) THEN
	Convert_LINT_TO_WORD := INCOMPATIBLE;
	RETURN;
END_IF

out := converted;

END_FUNCTION

// ---- Functions/Converters/LREAL_TO_/Convert_LREAL_TO_.TcPOU
FUNCTION Convert_LREAL_TO_ : Hresult
VAR_INPUT
	in : LREAL;
	out : ANY;
END_VAR
VAR
	convertResult : HRESULT := INCOMPATIBLE;
	convertAddress : PVOID;
	_BOOL : BOOL;
	_BYTE : BYTE;
	_DATE : DATE;
	_DINT : DINT;
	_DT : DT;
	_DWORD : DWORD;
	_INT : INT;
	_LINT : LINT;
	_LREAL : LREAL;
	_LWORD : LWORD;
	_REAL : REAL;
	_SINT : SINT;
	_STRING : STRING;
	_TIME : TIME;
	_TOD : TOD;
	_UDINT : UDINT;
	_UINT : UINT;
	_ULINT : ULINT;
	_USINT : USINT;
	_WORD : WORD;
END_VAR

CASE out.TypeClass OF
	
	__SYSTEM.TYPE_CLASS.TYPE_BOOL:
	
		convertResult := Convert_LREAL_TO_BOOL(in, _BOOL);
		IF SUCCEEDED(convertResult) THEN
			convertAddress := ADR(_BOOL);
		END_IF

	__SYSTEM.TYPE_CLASS.TYPE_BYTE:
	
		convertResult := Convert_LREAL_TO_BYTE(in, _BYTE);
		IF SUCCEEDED(convertResult) THEN
			convertAddress := ADR(_BYTE);
		END_IF

	__SYSTEM.TYPE_CLASS.TYPE_DATE:
	
		convertResult := Convert_LREAL_TO_DATE(in, _DATE);
		IF SUCCEEDED(convertResult) THEN
			convertAddress := ADR(_DATE);
		END_IF

	__SYSTEM.TYPE_CLASS.TYPE_DINT:
	
		convertResult := Convert_LREAL_TO_DINT(in, _DINT);
		IF SUCCEEDED(convertResult) THEN
			convertAddress := ADR(_DINT);
		END_IF

	__SYSTEM.TYPE_CLASS.TYPE_DATEANDTIME:
	
		convertResult := Convert_LREAL_TO_DT(in, _DT);
		IF SUCCEEDED(convertResult) THEN
			convertAddress := ADR(_DT);
		END_IF

	__SYSTEM.TYPE_CLASS.TYPE_DWORD:
	
		convertResult := Convert_LREAL_TO_DWORD(in, _DWORD);
		IF SUCCEEDED(convertResult) THEN
			convertAddress := ADR(_DWORD);
		END_IF

	__SYSTEM.TYPE_CLASS.TYPE_INT:
	
		convertResult := Convert_LREAL_TO_INT(in, _INT);
		IF SUCCEEDED(convertResult) THEN
			convertAddress := ADR(_INT);
		END_IF

	__SYSTEM.TYPE_CLASS.TYPE_LINT:
	
		convertResult := Convert_LREAL_TO_LINT(in, _LINT);
		IF SUCCEEDED(convertResult) THEN
			convertAddress := ADR(_LINT);
		END_IF

	__SYSTEM.TYPE_CLASS.TYPE_LREAL:
	
		convertResult := Convert_LREAL_TO_LREAL(in, _LREAL);
		IF SUCCEEDED(convertResult) THEN
			convertAddress := ADR(_LREAL);
		END_IF

	__SYSTEM.TYPE_CLASS.TYPE_LWORD:
	
		convertResult := Convert_LREAL_TO_LWORD(in, _LWORD);
		IF SUCCEEDED(convertResult) THEN
			convertAddress := ADR(_LWORD);
		END_IF

	__SYSTEM.TYPE_CLASS.TYPE_REAL:
	
		convertResult := Convert_LREAL_TO_REAL(in, _REAL);
		IF SUCCEEDED(convertResult) THEN
			convertAddress := ADR(_REAL);
		END_IF

	__SYSTEM.TYPE_CLASS.TYPE_SINT:
	
		convertResult := Convert_LREAL_TO_SINT(in, _SINT);
		IF SUCCEEDED(convertResult) THEN
			convertAddress := ADR(_SINT);
		END_IF

	__SYSTEM.TYPE_CLASS.TYPE_STRING:
	
		convertResult := Convert_LREAL_TO_STRING(in, _STRING);
		IF SUCCEEDED(convertResult) THEN
			convertAddress := ADR(_STRING);
		END_IF

	__SYSTEM.TYPE_CLASS.TYPE_TIME:
	
		convertResult := Convert_LREAL_TO_TIME(in, _TIME);
		IF SUCCEEDED(convertResult) THEN
			convertAddress := ADR(_TIME);
		END_IF

	__SYSTEM.TYPE_CLASS.TYPE_TIMEOFDAY:
	
		convertResult := Convert_LREAL_TO_TOD(in, _TOD);
		IF SUCCEEDED(convertResult) THEN
			convertAddress := ADR(_TOD);
		END_IF

	__SYSTEM.TYPE_CLASS.TYPE_UDINT:
	
		convertResult := Convert_LREAL_TO_UDINT(in, _UDINT);
		IF SUCCEEDED(convertResult) THEN
			convertAddress := ADR(_UDINT);
		END_IF

	__SYSTEM.TYPE_CLASS.TYPE_UINT:
	
		convertResult := Convert_LREAL_TO_UINT(in, _UINT);
		IF SUCCEEDED(convertResult) THEN
			convertAddress := ADR(_UINT);
		END_IF

	__SYSTEM.TYPE_CLASS.TYPE_ULINT:
	
		convertResult := Convert_LREAL_TO_ULINT(in, _ULINT);
		IF SUCCEEDED(convertResult) THEN
			convertAddress := ADR(_ULINT);
		END_IF

	__SYSTEM.TYPE_CLASS.TYPE_USINT:
	
		convertResult := Convert_LREAL_TO_USINT(in, _USINT);
		IF SUCCEEDED(convertResult) THEN
			convertAddress := ADR(_USINT);
		END_IF

	__SYSTEM.TYPE_CLASS.TYPE_WORD:
	
		convertResult := Convert_LREAL_TO_WORD(in, _WORD);
		IF SUCCEEDED(convertResult) THEN
			convertAddress := ADR(_WORD);
		END_IF

END_CASE

IF SUCCEEDED(convertResult) THEN
	memcpy(out.pValue,convertAddress,DINT_TO_UDINT(out.diSize));
END_IF

Convert_LREAL_TO_ := convertResult;

END_FUNCTION

// ---- Functions/Converters/LREAL_TO_/Convert_LREAL_TO_BOOL.TcPOU
FUNCTION Convert_LREAL_TO_BOOL : Hresult
VAR_INPUT
	in : LREAL;
	out : REFERENCE TO BOOL;
END_VAR
VAR
	converted : BOOL;
END_VAR

converted := LREAL_TO_BOOL(in);

IF (BOOL_TO_LREAL(converted) <> in) THEN
	Convert_LREAL_TO_BOOL := INCOMPATIBLE;
	RETURN;
END_IF

out := converted;

END_FUNCTION

// ---- Functions/Converters/LREAL_TO_/Convert_LREAL_TO_BYTE.TcPOU
FUNCTION Convert_LREAL_TO_BYTE : Hresult
VAR_INPUT
	in : LREAL;
	out : REFERENCE TO BYTE;
END_VAR
VAR
	converted : BYTE;
END_VAR

converted := LREAL_TO_BYTE(in);

IF (BYTE_TO_LREAL(converted) <> in) THEN
	Convert_LREAL_TO_BYTE := INCOMPATIBLE;
	RETURN;
END_IF

out := converted;

END_FUNCTION

// ---- Functions/Converters/LREAL_TO_/Convert_LREAL_TO_DATE.TcPOU
FUNCTION Convert_LREAL_TO_DATE : Hresult
VAR_INPUT
	in : LREAL;
	out : REFERENCE TO DATE;
END_VAR
VAR
	converted : DATE;
END_VAR

converted := LREAL_TO_DATE(in);

IF (DATE_TO_LREAL(converted) <> in) THEN
	Convert_LREAL_TO_DATE := INCOMPATIBLE;
	RETURN;
END_IF

out := converted;

END_FUNCTION

// ---- Functions/Converters/LREAL_TO_/Convert_LREAL_TO_DT.TcPOU
FUNCTION Convert_LREAL_TO_DT : Hresult
VAR_INPUT
	in : LREAL;
	out : REFERENCE TO DT;
END_VAR
VAR
	converted : DT;
END_VAR

converted := LREAL_TO_DT(in);

IF (DT_TO_LREAL(converted) <> in) THEN
	Convert_LREAL_TO_DT := INCOMPATIBLE;
	RETURN;
END_IF

out := converted;

END_FUNCTION

// ---- Functions/Converters/LREAL_TO_/Convert_LREAL_TO_DWORD.TcPOU
FUNCTION Convert_LREAL_TO_DWORD : Hresult
VAR_INPUT
	in : LREAL;
	out : REFERENCE TO DWORD;
END_VAR
VAR
	converted : DWORD;
END_VAR

converted := LREAL_TO_DWORD(in);

IF (DWORD_TO_LREAL(converted) <> in) THEN
	Convert_LREAL_TO_DWORD := INCOMPATIBLE;
	RETURN;
END_IF

out := converted;

END_FUNCTION

// ---- Functions/Converters/LREAL_TO_/Convert_LREAL_TO_INT.TcPOU
FUNCTION Convert_LREAL_TO_INT : Hresult
VAR_INPUT
	in : LREAL;
	out : REFERENCE TO INT;
END_VAR
VAR
	converted : INT;
END_VAR

converted := LREAL_TO_INT(in);

IF (INT_TO_LREAL(converted) <> in) THEN
	Convert_LREAL_TO_INT := INCOMPATIBLE;
	RETURN;
END_IF

out := converted;

END_FUNCTION

// ---- Functions/Converters/LREAL_TO_/Convert_LREAL_TO_LWORD.TcPOU
FUNCTION Convert_LREAL_TO_LWORD : Hresult
VAR_INPUT
	in : LREAL;
	out : REFERENCE TO LWORD;
END_VAR
VAR
	converted : LWORD;
END_VAR

converted := LREAL_TO_LWORD(in);

IF (LWORD_TO_LREAL(converted) <> in) THEN
	Convert_LREAL_TO_LWORD := INCOMPATIBLE;
	RETURN;
END_IF

out := converted;

END_FUNCTION

// ---- Functions/Converters/LREAL_TO_/Convert_LREAL_TO_TIME.TcPOU
FUNCTION Convert_LREAL_TO_TIME : Hresult
VAR_INPUT
	in : LREAL;
	out : REFERENCE TO TIME;
END_VAR
VAR
	converted : TIME;
END_VAR

converted := LREAL_TO_TIME(in);

IF (TIME_TO_LREAL(converted) <> in) THEN
	Convert_LREAL_TO_TIME := INCOMPATIBLE;
	RETURN;
END_IF

out := converted;

END_FUNCTION

// ---- Functions/Converters/LREAL_TO_/Convert_LREAL_TO_UINT.TcPOU
FUNCTION Convert_LREAL_TO_UINT : Hresult
VAR_INPUT
	in : LREAL;
	out : REFERENCE TO UINT;
END_VAR
VAR
	converted : UINT;
END_VAR

converted := LREAL_TO_UINT(in);

IF (UINT_TO_LREAL(converted) <> in) THEN
	Convert_LREAL_TO_UINT := INCOMPATIBLE;
	RETURN;
END_IF

out := converted;

END_FUNCTION

// ---- Functions/Converters/LREAL_TO_/Convert_LREAL_TO_ULINT.TcPOU
FUNCTION Convert_LREAL_TO_ULINT : Hresult
VAR_INPUT
	in : LREAL;
	out : REFERENCE TO ULINT;
END_VAR
VAR
	converted : ULINT;
END_VAR

converted := LREAL_TO_ULINT(in);

IF (ULINT_TO_LREAL(converted) <> in) THEN
	Convert_LREAL_TO_ULINT := INCOMPATIBLE;
	RETURN;
END_IF

out := converted;

END_FUNCTION

// ---- Functions/Converters/LREAL_TO_/Convert_LREAL_TO_USINT.TcPOU
FUNCTION Convert_LREAL_TO_USINT : Hresult
VAR_INPUT
	in : LREAL;
	out : REFERENCE TO USINT;
END_VAR
VAR
	converted : USINT;
END_VAR

converted := LREAL_TO_USINT(in);

IF (USINT_TO_LREAL(converted) <> in) THEN
	Convert_LREAL_TO_USINT := INCOMPATIBLE;
	RETURN;
END_IF

out := converted;

END_FUNCTION

// ---- Functions/Converters/LREAL_TO_/Convert_LREAL_TO_WORD.TcPOU
FUNCTION Convert_LREAL_TO_WORD : Hresult
VAR_INPUT
	in : LREAL;
	out : REFERENCE TO WORD;
END_VAR
VAR
	converted : WORD;
END_VAR

converted := LREAL_TO_WORD(in);

IF (WORD_TO_LREAL(converted) <> in) THEN
	Convert_LREAL_TO_WORD := INCOMPATIBLE;
	RETURN;
END_IF

out := converted;

END_FUNCTION

// ---- Functions/Converters/LWORD_TO_/Convert_LWORD_TO_BOOL.TcPOU
FUNCTION Convert_LWORD_TO_BOOL : Hresult
VAR_INPUT
	in : LWORD;
	out : REFERENCE TO BOOL;
END_VAR
VAR
	converted : BOOL;
END_VAR

converted := LWORD_TO_BOOL(in);

IF (BOOL_TO_LWORD(converted) <> in) THEN
	Convert_LWORD_TO_BOOL := INCOMPATIBLE;
	RETURN;
END_IF

out := converted;

END_FUNCTION

// ---- Functions/Converters/LWORD_TO_/Convert_LWORD_TO_LINT.TcPOU
FUNCTION Convert_LWORD_TO_LINT : Hresult
VAR_INPUT
	in : LWORD;
	out : REFERENCE TO LINT;
END_VAR
VAR
	converted : LINT;
END_VAR

converted := LWORD_TO_LINT(in);

IF (LINT_TO_LWORD(converted) <> in) THEN
	Convert_LWORD_TO_LINT := INCOMPATIBLE;
	RETURN;
END_IF

out := converted;

END_FUNCTION

// ---- Functions/Converters/LWORD_TO_/Convert_LWORD_TO_SINT.TcPOU
FUNCTION Convert_LWORD_TO_SINT : Hresult
VAR_INPUT
	in : LWORD;
	out : REFERENCE TO SINT;
END_VAR
VAR
	converted : SINT;
END_VAR

converted := LWORD_TO_SINT(in);

IF (SINT_TO_LWORD(converted) <> in) THEN
	Convert_LWORD_TO_SINT := INCOMPATIBLE;
	RETURN;
END_IF

out := converted;

END_FUNCTION

// ---- Functions/Converters/LWORD_TO_/Convert_LWORD_TO_STRING.TcPOU
FUNCTION Convert_LWORD_TO_STRING : Hresult
VAR_INPUT
	in : LWORD;
	out : REFERENCE TO STRING;
END_VAR
VAR
	converted : STRING;
END_VAR

converted := LWORD_TO_STRING(in);

IF (STRING_TO_LWORD(converted) <> in) THEN
	Convert_LWORD_TO_STRING := INCOMPATIBLE;
	RETURN;
END_IF

out := converted;

END_FUNCTION

// ---- Functions/Converters/LWORD_TO_/Convert_LWORD_TO_TIME.TcPOU
FUNCTION Convert_LWORD_TO_TIME : Hresult
VAR_INPUT
	in : LWORD;
	out : REFERENCE TO TIME;
END_VAR
VAR
	converted : TIME;
END_VAR

converted := LWORD_TO_TIME(in);

IF (TIME_TO_LWORD(converted) <> in) THEN
	Convert_LWORD_TO_TIME := INCOMPATIBLE;
	RETURN;
END_IF

out := converted;

END_FUNCTION

// ---- Functions/Converters/LWORD_TO_/Convert_LWORD_TO_UDINT.TcPOU
FUNCTION Convert_LWORD_TO_UDINT : Hresult
VAR_INPUT
	in : LWORD;
	out : REFERENCE TO UDINT;
END_VAR
VAR
	converted : UDINT;
END_VAR

converted := LWORD_TO_UDINT(in);

IF (UDINT_TO_LWORD(converted) <> in) THEN
	Convert_LWORD_TO_UDINT := INCOMPATIBLE;
	RETURN;
END_IF

out := converted;

END_FUNCTION

// ---- Functions/Converters/LWORD_TO_/Convert_LWORD_TO_UINT.TcPOU
FUNCTION Convert_LWORD_TO_UINT : Hresult
VAR_INPUT
	in : LWORD;
	out : REFERENCE TO UINT;
END_VAR
VAR
	converted : UINT;
END_VAR

converted := LWORD_TO_UINT(in);

IF (UINT_TO_LWORD(converted) <> in) THEN
	Convert_LWORD_TO_UINT := INCOMPATIBLE;
	RETURN;
END_IF

out := converted;

END_FUNCTION

// ---- Functions/Converters/LWORD_TO_/Convert_LWORD_TO_USINT.TcPOU
FUNCTION Convert_LWORD_TO_USINT : Hresult
VAR_INPUT
	in : LWORD;
	out : REFERENCE TO USINT;
END_VAR
VAR
	converted : USINT;
END_VAR

converted := LWORD_TO_USINT(in);

IF (USINT_TO_LWORD(converted) <> in) THEN
	Convert_LWORD_TO_USINT := INCOMPATIBLE;
	RETURN;
END_IF

out := converted;

END_FUNCTION

// ---- Functions/Converters/REAL_TO_/Convert_REAL_TO_.TcPOU
FUNCTION Convert_REAL_TO_ : Hresult
VAR_INPUT
	in : REAL;
	out : ANY;
END_VAR
VAR
	convertResult : HRESULT := INCOMPATIBLE;
	convertAddress : PVOID;
	_BOOL : BOOL;
	_BYTE : BYTE;
	_DATE : DATE;
	_DINT : DINT;
	_DT : DT;
	_DWORD : DWORD;
	_INT : INT;
	_LINT : LINT;
	_LREAL : LREAL;
	_LWORD : LWORD;
	_REAL : REAL;
	_SINT : SINT;
	_STRING : STRING;
	_TIME : TIME;
	_TOD : TOD;
	_UDINT : UDINT;
	_UINT : UINT;
	_ULINT : ULINT;
	_USINT : USINT;
	_WORD : WORD;
END_VAR

CASE out.TypeClass OF
	
	__SYSTEM.TYPE_CLASS.TYPE_BOOL:
	
		convertResult := Convert_REAL_TO_BOOL(in, _BOOL);
		IF SUCCEEDED(convertResult) THEN
			convertAddress := ADR(_BOOL);
		END_IF

	__SYSTEM.TYPE_CLASS.TYPE_BYTE:
	
		convertResult := Convert_REAL_TO_BYTE(in, _BYTE);
		IF SUCCEEDED(convertResult) THEN
			convertAddress := ADR(_BYTE);
		END_IF

	__SYSTEM.TYPE_CLASS.TYPE_DATE:
	
		convertResult := Convert_REAL_TO_DATE(in, _DATE);
		IF SUCCEEDED(convertResult) THEN
			convertAddress := ADR(_DATE);
		END_IF

	__SYSTEM.TYPE_CLASS.TYPE_DINT:
	
		convertResult := Convert_REAL_TO_DINT(in, _DINT);
		IF SUCCEEDED(convertResult) THEN
			convertAddress := ADR(_DINT);
		END_IF

	__SYSTEM.TYPE_CLASS.TYPE_DATEANDTIME:
	
		convertResult := Convert_REAL_TO_DT(in, _DT);
		IF SUCCEEDED(convertResult) THEN
			convertAddress := ADR(_DT);
		END_IF

	__SYSTEM.TYPE_CLASS.TYPE_DWORD:
	
		convertResult := Convert_REAL_TO_DWORD(in, _DWORD);
		IF SUCCEEDED(convertResult) THEN
			convertAddress := ADR(_DWORD);
		END_IF

	__SYSTEM.TYPE_CLASS.TYPE_INT:
	
		convertResult := Convert_REAL_TO_INT(in, _INT);
		IF SUCCEEDED(convertResult) THEN
			convertAddress := ADR(_INT);
		END_IF

	__SYSTEM.TYPE_CLASS.TYPE_LINT:
	
		convertResult := Convert_REAL_TO_LINT(in, _LINT);
		IF SUCCEEDED(convertResult) THEN
			convertAddress := ADR(_LINT);
		END_IF

	__SYSTEM.TYPE_CLASS.TYPE_LREAL:
	
		convertResult := Convert_REAL_TO_LREAL(in, _LREAL);
		IF SUCCEEDED(convertResult) THEN
			convertAddress := ADR(_LREAL);
		END_IF

	__SYSTEM.TYPE_CLASS.TYPE_LWORD:
	
		convertResult := Convert_REAL_TO_LWORD(in, _LWORD);
		IF SUCCEEDED(convertResult) THEN
			convertAddress := ADR(_LWORD);
		END_IF

	__SYSTEM.TYPE_CLASS.TYPE_REAL:
	
		convertResult := Convert_REAL_TO_REAL(in, _REAL);
		IF SUCCEEDED(convertResult) THEN
			convertAddress := ADR(_REAL);
		END_IF

	__SYSTEM.TYPE_CLASS.TYPE_SINT:
	
		convertResult := Convert_REAL_TO_SINT(in, _SINT);
		IF SUCCEEDED(convertResult) THEN
			convertAddress := ADR(_SINT);
		END_IF

	__SYSTEM.TYPE_CLASS.TYPE_STRING:
	
		convertResult := Convert_REAL_TO_STRING(in, _STRING);
		IF SUCCEEDED(convertResult) THEN
			convertAddress := ADR(_STRING);
		END_IF

	__SYSTEM.TYPE_CLASS.TYPE_TIME:
	
		convertResult := Convert_REAL_TO_TIME(in, _TIME);
		IF SUCCEEDED(convertResult) THEN
			convertAddress := ADR(_TIME);
		END_IF

	__SYSTEM.TYPE_CLASS.TYPE_TIMEOFDAY:
	
		convertResult := Convert_REAL_TO_TOD(in, _TOD);
		IF SUCCEEDED(convertResult) THEN
			convertAddress := ADR(_TOD);
		END_IF

	__SYSTEM.TYPE_CLASS.TYPE_UDINT:
	
		convertResult := Convert_REAL_TO_UDINT(in, _UDINT);
		IF SUCCEEDED(convertResult) THEN
			convertAddress := ADR(_UDINT);
		END_IF

	__SYSTEM.TYPE_CLASS.TYPE_UINT:
	
		convertResult := Convert_REAL_TO_UINT(in, _UINT);
		IF SUCCEEDED(convertResult) THEN
			convertAddress := ADR(_UINT);
		END_IF

	__SYSTEM.TYPE_CLASS.TYPE_ULINT:
	
		convertResult := Convert_REAL_TO_ULINT(in, _ULINT);
		IF SUCCEEDED(convertResult) THEN
			convertAddress := ADR(_ULINT);
		END_IF

	__SYSTEM.TYPE_CLASS.TYPE_USINT:
	
		convertResult := Convert_REAL_TO_USINT(in, _USINT);
		IF SUCCEEDED(convertResult) THEN
			convertAddress := ADR(_USINT);
		END_IF

	__SYSTEM.TYPE_CLASS.TYPE_WORD:
	
		convertResult := Convert_REAL_TO_WORD(in, _WORD);
		IF SUCCEEDED(convertResult) THEN
			convertAddress := ADR(_WORD);
		END_IF

END_CASE

IF SUCCEEDED(convertResult) THEN
	memcpy(out.pValue,convertAddress,DINT_TO_UDINT(out.diSize));
END_IF

Convert_REAL_TO_ := convertResult;

END_FUNCTION

// ---- Functions/Converters/REAL_TO_/Convert_REAL_TO_BYTE.TcPOU
FUNCTION Convert_REAL_TO_BYTE : Hresult
VAR_INPUT
	in : REAL;
	out : REFERENCE TO BYTE;
END_VAR
VAR
	converted : BYTE;
END_VAR

converted := REAL_TO_BYTE(in);

IF (BYTE_TO_REAL(converted) <> in) THEN
	Convert_REAL_TO_BYTE := INCOMPATIBLE;
	RETURN;
END_IF

out := converted;

END_FUNCTION

// ---- Functions/Converters/REAL_TO_/Convert_REAL_TO_DATE.TcPOU
FUNCTION Convert_REAL_TO_DATE : Hresult
VAR_INPUT
	in : REAL;
	out : REFERENCE TO DATE;
END_VAR
VAR
	converted : DATE;
END_VAR

converted := REAL_TO_DATE(in);

IF (DATE_TO_REAL(converted) <> in) THEN
	Convert_REAL_TO_DATE := INCOMPATIBLE;
	RETURN;
END_IF

out := converted;

END_FUNCTION

// ---- Functions/Converters/REAL_TO_/Convert_REAL_TO_DINT.TcPOU
FUNCTION Convert_REAL_TO_DINT : Hresult
VAR_INPUT
	in : REAL;
	out : REFERENCE TO DINT;
END_VAR
VAR
	converted : DINT;
END_VAR

converted := REAL_TO_DINT(in);

IF (DINT_TO_REAL(converted) <> in) THEN
	Convert_REAL_TO_DINT := INCOMPATIBLE;
	RETURN;
END_IF

out := converted;

END_FUNCTION

// ---- Functions/Converters/REAL_TO_/Convert_REAL_TO_DWORD.TcPOU
FUNCTION Convert_REAL_TO_DWORD : Hresult
VAR_INPUT
	in : REAL;
	out : REFERENCE TO DWORD;
END_VAR
VAR
	converted : DWORD;
END_VAR

converted := REAL_TO_DWORD(in);

IF (DWORD_TO_REAL(converted) <> in) THEN
	Convert_REAL_TO_DWORD := INCOMPATIBLE;
	RETURN;
END_IF

out := converted;

END_FUNCTION

// ---- Functions/Converters/REAL_TO_/Convert_REAL_TO_LINT.TcPOU
FUNCTION Convert_REAL_TO_LINT : Hresult
VAR_INPUT
	in : REAL;
	out : REFERENCE TO LINT;
END_VAR
VAR
	converted : LINT;
END_VAR

converted := REAL_TO_LINT(in);

IF (LINT_TO_REAL(converted) <> in) THEN
	Convert_REAL_TO_LINT := INCOMPATIBLE;
	RETURN;
END_IF

out := converted;

END_FUNCTION

// ---- Functions/Converters/REAL_TO_/Convert_REAL_TO_LWORD.TcPOU
FUNCTION Convert_REAL_TO_LWORD : Hresult
VAR_INPUT
	in : REAL;
	out : REFERENCE TO LWORD;
END_VAR
VAR
	converted : LWORD;
END_VAR

converted := REAL_TO_LWORD(in);

IF (LWORD_TO_REAL(converted) <> in) THEN
	Convert_REAL_TO_LWORD := INCOMPATIBLE;
	RETURN;
END_IF

out := converted;

END_FUNCTION

// ---- Functions/Converters/REAL_TO_/Convert_REAL_TO_STRING.TcPOU
FUNCTION Convert_REAL_TO_STRING : Hresult
VAR_INPUT
	in : REAL;
	out : REFERENCE TO STRING;
END_VAR
VAR
	converted : STRING;
END_VAR

converted := REAL_TO_STRING(in);

IF (STRING_TO_REAL(converted) <> in) THEN
	Convert_REAL_TO_STRING := INCOMPATIBLE;
	RETURN;
END_IF

out := converted;

END_FUNCTION

// ---- Functions/Disposable/F_SafeRelease.TcPOU
FUNCTION F_SafeRelease
VAR_INPUT
	Object : I_Disposable;
END_VAR

IF Object <> 0 THEN
	Object.Release();
END_IF

END_FUNCTION

// ---- _Internal/Collections/Collection.TcPOU
{attribute 'linkalways'} 
{attribute 'no_explicit_call' := 'This FB is a CLASS and must be accessed using methods or properties'}
{attribute 'enable_dynamic_creation'}
FUNCTION_BLOCK Collection
VAR
	head : I_CollectionNode;
END_VAR

PROPERTY PUBLIC Count : UDINT
GET
VAR
	currentCount : UDINT;
	currentNode : I_CollectionNode;
END_VAR
currentCount := 0;
currentNode := head;

WHILE currentNode <> 0 DO
	currentNode := currentNode.Next;
	currentCount := currentCount + 1;
END_WHILE;

Count := currentCount;
END_GET
END_PROPERTY

METHOD FB_exit : BOOL
VAR_INPUT
	bInCopyCode : BOOL; // if TRUE, the exit method is called for exiting an instance that is copied afterwards (online change).
END_VAR
VAR
	previousNode : I_CollectionNode;
	currentNode : I_CollectionNode;
END_VAR
currentNode := head;

WHILE currentNode <> 0 DO
	previousNode := currentNode;
	currentNode := previousNode.Next;
	
	previousNode.Destroy();
END_WHILE;
END_METHOD

METHOD PUBLIC GetByIndex : I_Collectable
VAR_INPUT
	Index : UDINT;
END_VAR
VAR
	currentNode : I_CollectionNode;
	counter : UDINT;
END_VAR
IF head = 0 THEN
	RETURN;
END_IF

currentNode := head;
counter := 0;

WHILE currentNode <> 0 DO
	
	IF counter = Index THEN
		GetByIndex := currentNode.Collectable;
		return;
	END_IF
	
	currentNode := currentNode.Next;
	counter := counter + 1;

END_WHILE;
END_METHOD

METHOD PUBLIC Insert
VAR_INPUT
	CollectableObject : I_Collectable;
END_VAR
VAR
	last : I_CollectionNode;
	pCollectionNode : POINTER TO CollectionNode;
END_VAR
pCollectionNode := __NEW(CollectionNode(Collectable := CollectableObject)); 

IF head = 0 THEN	
	head := pCollectionNode^; 
	RETURN;
END_IF

last := head; 

WHILE last.Next <> 0 DO
	last := last.next; 
END_WHILE;
	
last.next := pCollectionNode^;
END_METHOD

METHOD PUBLIC Remove
VAR_INPUT
	CollectableObject : I_Collectable;
END_VAR
VAR
	currentNode : I_CollectionNode;
	previousNode : I_CollectionNode;
END_VAR
IF head = 0 THEN
	RETURN;
END_IF

currentNode := head;

IF currentNode.Collectable = CollectableObject THEN
	
	head := currentNode.Next;
	currentNode.Next := 0;
	currentNode.Destroy();
	RETURN;
	
END_IF

WHILE currentNode <> 0 DO
	
	IF currentNode.Collectable = CollectableObject THEN
		EXIT;
	END_IF
	
	previousNode := currentNode;
	currentNode := currentNode.Next;

END_WHILE;

IF currentNode = 0 THEN
	RETURN;
END_IF

previousNode.Next := currentNode.Next;
currentNode.Next := 0;
currentNode.Destroy();
END_METHOD

METHOD PUBLIC RemoveByIndex
VAR_INPUT
	Index : UDINT;
END_VAR
VAR
	currentNode : I_CollectionNode;
	counter : UDINT;
	previousNode : I_CollectionNode;
END_VAR
IF head = 0 THEN
	RETURN;
END_IF

currentNode := head;

IF Index = 0 THEN
	
	head := currentNode.Next;
	currentNode.Next := 0;
	currentNode.Destroy();
	RETURN;
	
END_IF

counter := 0;

WHILE currentNode <> 0 DO
	
	IF counter = Index THEN
		EXIT;
	END_IF
	
